// ---- MTCS/Common/Widgets/OperatingButtonWidget.TcPOU
FUNCTION_BLOCK OperatingButtonWidget
VAR_INPUT
END_VAR
VAR_OUTPUT
    text : STRING;
    deactivate : BOOL;
END_VAR
VAR_IN_OUT
    status : OperatingStatus;
	process : ChangeOperatingStateProcess;
END_VAR
VAR
    do_request : BOOL := FALSE;
END_VAR

IF status.auto THEN
    text := 'Manual';
    process.set.state := OperatingStates.MANUAL;
    deactivate := process.statuses.enabledStatus.disabled;
ELSIF status.manual THEN
    text := 'Auto';
    process.set.state := OperatingStates.AUTO;
    deactivate := process.statuses.enabledStatus.disabled;
ELSE
    text := 'Auto';
    process.set.state := OperatingStates.MANUAL;
    deactivate := TRUE;
END_IF


IF do_request THEN
    process.request(state := process.set.state);
    do_request := FALSE;
END_IF

END_FUNCTION_BLOCK

// ---- MTCS/Common/Widgets/LockingButtonWidget.TcPOU
FUNCTION_BLOCK LockingButtonWidget
VAR_INPUT
END_VAR
VAR_OUTPUT
    text : STRING;
    deactivate : BOOL;
END_VAR
VAR_IN_OUT
    status : InitializationStatus;
	lock : Process;
	unlock : Process;
END_VAR
VAR
    do_request : BOOL := FALSE;
END_VAR

IF status.locked THEN
    text := 'Unlock';
    deactivate := unlock.statuses.enabledStatus.disabled;
    
    IF do_request THEN
        unlock.request();
        do_request := FALSE;
    END_IF

ELSIF status.initialized THEN
    text := 'Lock';
    deactivate := lock.statuses.enabledStatus.disabled;
    
    IF do_request THEN
        lock.request();
        do_request := FALSE;
    END_IF
ELSE
    text := 'Unlock';
    deactivate := TRUE;
    do_request := FALSE;
END_IF

END_FUNCTION_BLOCK

// ---- MTCS/Common/HelperCode/SystemToColor.TcPOU
FUNCTION SystemToColor : StatusColor
VAR_IN_OUT
    healthStatus : HealthStatus;
    busyStatus   : BusyStatus;
    initializationStatus : InitializationStatus;
    operatingStatus : OperatingStatus;
END_VAR
VAR_OUTPUT
END_VAR
VAR
END_VAR

IF initializationStatus.shutdown THEN
    SystemToColor.fg := Colors.BLACK;
    SystemToColor.bg := Colors.GRAY;
ELSIF initializationStatus.initializing THEN
    SystemToColor.fg := Colors.WHITE;
    SystemToColor.bg := Colors.BLUE;
ELSE
    IF healthStatus.good THEN
        IF busyStatus.busy THEN
            SystemToColor.fg := Colors.WHITE;
            SystemToColor.bg := Colors.BLUE;
        ELSE
            IF initializationStatus.locked OR operatingStatus.manual THEN
                SystemToColor.fg := Colors.WHITE;
                SystemToColor.bg := Colors.ORANGE;
            ELSE
                SystemToColor.fg := Colors.BLACK;
                SystemToColor.bg := Colors.GREEN;
			END_IF
        END_IF
    ELSIF healthStatus.bad THEN
        SystemToColor.fg := Colors.WHITE;
        SystemToColor.bg := Colors.RED;
    ELSIF healthStatus.warning THEN
        SystemToColor.fg := Colors.WHITE;
        SystemToColor.bg := Colors.ORANGE;
    ELSE
        SystemToColor.fg := Colors.BLACK;
        SystemToColor.bg := Colors.GRAY;
    END_IF
END_IF

END_FUNCTION

// ---- MTCS/Common/HelperCode/BusyToColor.TcPOU
FUNCTION BusyToColor : StatusColor
VAR_IN_OUT
    busyStatus : BusyStatus;
END_VAR
VAR_OUTPUT
END_VAR
VAR
END_VAR

IF busyStatus.idle THEN
    BusyToColor.fg := Colors.BLACK;
    BusyToColor.bg := Colors.GREEN;
ELSIF busyStatus.busy THEN
	BusyToColor.fg := Colors.WHITE;
	BusyToColor.bg := Colors.BLUE;
ELSE
	BusyToColor.fg := Colors.BLACK;
	BusyToColor.bg := Colors.GRAY;
END_IF

END_FUNCTION

// ---- MTCS/Common/HelperCode/DegToRad.TcPOU
FUNCTION DegToRad : LREAL
VAR_INPUT
    degrees : LREAL;
END_VAR
VAR
END_VAR

DegToRad := degrees / 180.0 * PI;

END_FUNCTION

// ---- MTCS/Common/HelperCode/MeasurementToString.TcPOU
FUNCTION_BLOCK MeasurementToString
VAR_INPUT
    value : LREAL;
    format : STRING;
    overrange : BOOL;
    underrange: BOOL;
    error : BOOL;
END_VAR
VAR_OUTPUT
    display : STRING;
    actualStatus : STRING;
END_VAR
VAR_IN_OUT
    alarmStatus : HiHiLoLoAlarmStatus;
    enabledStatus : EnabledStatus;
END_VAR
VAR
    _formatString : FB_FormatString;
END_VAR

// update the display and actualStatus
IF enabledStatus.enabled THEN
    IF overrange THEN
        display := '';
        actualStatus := 'Overrange';
    ELSIF underrange THEN
        display := '';
        actualStatus := 'Underrange';
    ELSIF error THEN
        display := '';
        actualStatus := 'Error';
    ELSE
        // update display:
        _formatString(sFormat := format, 
                      arg1    := F_LREAL(value),
                      sOut    => display);
        // update actualStatus:
        IF alarmStatus.disabled THEN
            actualStatus := 'Valid';
        ELSIF alarmStatus.ok THEN
            actualStatus := 'Valid and within range';
        ELSIF alarmStatus.hi THEN
            actualStatus := 'High!';
        ELSIF alarmStatus.hiHi THEN
            actualStatus := 'Critically high!';
        ELSIF alarmStatus.lo THEN
            actualStatus := 'Low!';
        ELSIF alarmStatus.loLo THEN
            actualStatus := 'Critically low!';
        ELSE
            actualStatus := display;
        END_IF
    END_IF
ELSIF enabledStatus.disabled THEN
    display := '';
    actualStatus := 'Disabled';
ELSE
    display := '';
    actualStatus := 'UNKNOWN';
END_IF

END_FUNCTION_BLOCK

// ---- MTCS/Common/HelperCode/MeasurementToStatus.TcPOU
FUNCTION_BLOCK MeasurementToStatus
VAR_INPUT
    overrange : BOOL;
    underrange: BOOL;
    error : BOOL;
END_VAR
VAR_OUTPUT
    actualStatus : STRING;
END_VAR
VAR_IN_OUT
    alarmStatus : HiHiLoLoAlarmStatus;
    enabledStatus : EnabledStatus;
END_VAR
VAR
END_VAR

// update the display and actualStatus
IF enabledStatus.enabled THEN
    IF overrange THEN
        actualStatus := 'Overrange';
    ELSIF underrange THEN
        actualStatus := 'Underrange';
    ELSIF error THEN
        actualStatus := 'Error';
    ELSE
        // update actualStatus:
        IF alarmStatus.disabled THEN
            actualStatus := 'Valid';
        ELSIF alarmStatus.ok THEN
            actualStatus := 'Valid and within range';
        ELSIF alarmStatus.hi THEN
            actualStatus := 'High!';
        ELSIF alarmStatus.hiHi THEN
            actualStatus := 'Critically high!';
        ELSIF alarmStatus.lo THEN
            actualStatus := 'Low!';
        ELSIF alarmStatus.loLo THEN
            actualStatus := 'Critically low!';
        ELSE
            actualStatus := 'UNKNOWN';
        END_IF
    END_IF
ELSIF enabledStatus.disabled THEN
    actualStatus := 'Disabled';
ELSE
    actualStatus := 'UNKNOWN';
END_IF

END_FUNCTION_BLOCK

// ---- MTCS/Common/HelperCode/RadToDeg.TcPOU
FUNCTION RadToDeg : LREAL
VAR_INPUT
    radians : LREAL;
END_VAR
VAR
END_VAR

RadToDeg := radians / PI * 180.0;

END_FUNCTION

// ---- MTCS/Common/StateMachines/AngularVelocity.TcPOU
FUNCTION_BLOCK AngularVelocity EXTENDS SM_AngularVelocity
VAR_INPUT
END_VAR
VAR_OUTPUT
END_VAR
VAR
    _testVar : INT;
END_VAR

SUPER^();

END_FUNCTION_BLOCK

// ---- MTCS/Common/StateMachines/AngularAcceleration.TcPOU
FUNCTION_BLOCK AngularAcceleration EXTENDS SM_AngularAcceleration
VAR_INPUT
END_VAR
VAR_OUTPUT
END_VAR
VAR
    _testVar : INT;
END_VAR

SUPER^();

END_FUNCTION_BLOCK

// ---- MTCS/Common/StateMachines/AverageCurrent.TcPOU
FUNCTION_BLOCK AverageCurrent EXTENDS SM_AverageCurrent
VAR_INPUT
    noOfSamples : UINT := 100;
    ctrlTimeMultiplier : UINT := 1;
END_VAR
VAR_OUTPUT
END_VAR
VAR
    _ctrl_moving_avg : FB_CTRL_MOVING_AVERAGE;
    _params : ST_CTRL_MOVING_AVERAGE_PARAMS;
    _array : ARRAY [1..100] OF LREAL;
END_VAR

_params.nSamplesToFilter  := noOfSamples;
_params.tCtrlCycleTime    := GLOBAL.config.PLC_CTRL_TIME * ctrlTimeMultiplier;

_ctrl_moving_avg(
    fIn             := SUPER^.newAmpsValue,
    fManSyncValue   := 0.0,
    bSync           := FALSE,
    eMode           := E_CTRL_MODE.eCTRL_MODE_ACTIVE,
    bHold           := FALSE,
    stParams        := _params);

SUPER^(newAmpsValue := _ctrl_moving_avg.fOut);

METHOD FB_init : BOOL
VAR_INPUT
	bInitRetains : BOOL; // if TRUE, the retain variables are initialized (warm start / cold start)
	bInCopyCode : BOOL;  // if TRUE, the instance afterwards gets moved into the copy code (online change)
END_VAR
_params.tTaskCycleTime    := GLOBAL.config.PLC_TASK_TIME;
_params.pWorkArray_ADR    := ADR(_array);
_params.nWorkArray_SIZEOF := SIZEOF(_array);
END_METHOD

END_FUNCTION_BLOCK

// ---- MTCS/Common/StateMachines/AX52XXDrive.TcPOU
FUNCTION_BLOCK AX52XXDrive EXTENDS SM_AX52XXDrive
VAR_INPUT
END_VAR
VAR_OUTPUT
END_VAR
VAR
    _internal : INT; // if no variable is present, the symbols of the superclass are not visible in the OPC UA address space
END_VAR

SUPER^();

END_FUNCTION_BLOCK

// ---- MTCS/Common/StateMachines/BaseProcess.TcPOU
FUNCTION_BLOCK BaseProcess EXTENDS SM_BaseProcess (* default process *)
VAR_INPUT
	_state : INT; // internal state, may or may not be used
END_VAR
VAR_OUTPUT
END_VAR
VAR
END_VAR

// we make it easy for ourselves: every time the process is idle, we reset the startedStatus
IF statuses.busyStatus.idle THEN
	statuses.startedStatus(isStarted := FALSE);
END_IF

_update();

METHOD isIdle : BOOL
VAR_INPUT
END_VAR
isIdle := statuses.busyStatus.idle;
END_METHOD

METHOD _update
VAR_INPUT
END_VAR

IF actualStatus = '' THEN
    IF statuses.enabledStatus.disabled THEN
        actualStatus := '';
    ELSIF statuses.enabledStatus.enabled THEN
        IF statuses.healthStatus.good THEN
            IF statuses.busyStatus.busy THEN
                actualStatus := 'Busy';
            ELSIF statuses.busyStatus.idle THEN
                actualStatus := 'Idle';
            ELSE
                actualStatus := 'Good but UNKNOWN';
            END_IF
        ELSIF statuses.healthStatus.bad THEN
            IF statuses.busyStatus.busy THEN
                actualStatus := 'Error (busy)';
            ELSIF statuses.busyStatus.idle THEN
                actualStatus := 'Error';
            ELSE
                actualStatus := 'Bad but UNKNOWN';
            END_IF
        END_IF
    END_IF
END_IF

SUPER^();
END_METHOD

METHOD setBad
VAR_INPUT
END_VAR
statuses.healthStatus(isGood := FALSE);
END_METHOD

METHOD resetIfIdle
VAR_INPUT
END_VAR
IF statuses.busyStatus.idle  THEN
    
    statuses.healthStatus(isGood := TRUE, hasWarning := FALSE);
    setActualStatus('Idle');
    setFinished();
    
END_IF
END_METHOD

METHOD setBusy
VAR_INPUT
END_VAR
statuses.busyStatus(isBusy := TRUE);
END_METHOD

METHOD setFinished
VAR_INPUT
END_VAR
statuses.busyStatus(isBusy := FALSE);
statuses.startedStatus(isStarted := FALSE);
END_METHOD

METHOD setStarted
VAR_INPUT
END_VAR
statuses.startedStatus(isStarted := TRUE);
END_METHOD

METHOD isBusy : BOOL
VAR_INPUT
END_VAR
isBusy := statuses.busyStatus.busy;
END_METHOD

METHOD setActualStatus
VAR_INPUT
    msg : STRING;
END_VAR
actualStatus := msg;
END_METHOD

METHOD reset
VAR_INPUT
END_VAR
statuses.healthStatus(isGood := TRUE, hasWarning := FALSE);
statuses.busyStatus(isBusy := FALSE);
setActualStatus('Idle');
setFinished();
END_METHOD

METHOD setGood
VAR_INPUT
END_VAR
statuses.healthStatus(isGood := TRUE);
END_METHOD

METHOD isGood : BOOL
VAR_INPUT
END_VAR
isGood := statuses.healthStatus.good;
END_METHOD

METHOD FB_init : BOOL
VAR_INPUT
	bInitRetains : BOOL; // if TRUE, the retain variables are initialized (warm start / cold start)
	bInCopyCode : BOOL;  // if TRUE, the instance afterwards gets moved into the copy code (online change)
END_VAR
statuses.busyStatus(isBusy := FALSE);
statuses.startedStatus(isStarted := FALSE);
statuses.healthStatus(isGood := TRUE);
END_METHOD

METHOD isStarted : BOOL
VAR_INPUT
END_VAR
isStarted := statuses.startedStatus.started;
END_METHOD

END_FUNCTION_BLOCK

// ---- MTCS/Common/StateMachines/BaseXmlDataSrvProcess.TcPOU
FUNCTION_BLOCK BaseXmlDataSrvProcess EXTENDS SM_BaseMcProcess
VAR_INPUT
END_VAR
VAR_OUTPUT
END_VAR
VAR
	testVar3 : BOOL;
END_VAR

SUPER^();

END_FUNCTION_BLOCK

// ---- MTCS/Common/StateMachines/CANopenBus.TcPOU
FUNCTION_BLOCK CANopenBus EXTENDS SM_CANopenBus
VAR_INPUT
END_VAR
VAR_OUTPUT
END_VAR
VAR
    testVar : INT;
END_VAR

//IF GLOBAL.CONFIG.SIMULATION_ACTIVE THEN
//    SUPER^.infoData := 8;
//    SUPER^.wcState := FALSE;
//END_IF

SUPER^();

IF error = 0 THEN
    actualStatus := 'No errors';
ELSE
    actualStatus := CONCAT(USINT_TO_STRING(error), ' boxes have errors');
END_IF

END_FUNCTION_BLOCK

// ---- MTCS/Common/StateMachines/CurrentMeasurement.TcPOU
FUNCTION_BLOCK CurrentMeasurement EXTENDS SM_CurrentMeasurement
VAR_INPUT
END_VAR
VAR_OUTPUT
END_VAR
VAR
    testVar : INT;
END_VAR

SUPER^();

END_FUNCTION_BLOCK

// ---- MTCS/Common/StateMachines/GForce.TcPOU
FUNCTION_BLOCK GForce EXTENDS SM_GForce
VAR_INPUT
END_VAR
VAR_OUTPUT
END_VAR
VAR
    _testVar : INT;
END_VAR

SUPER^();

END_FUNCTION_BLOCK

// ---- MTCS/Common/StateMachines/LinearPositionMeasurement16.TcPOU
FUNCTION_BLOCK LinearPositionMeasurement16 EXTENDS SM_LinearPositionMeasurement16
VAR_INPUT
END_VAR
VAR_OUTPUT
END_VAR
VAR
    noOfSamples : UINT := 100;
    _toStatus : MeasurementToStatus;
	_executeMovingAverage : BOOL;
    _ctrl_moving_avg : FB_CTRL_MOVING_AVERAGE;
    _params : ST_CTRL_MOVING_AVERAGE_PARAMS;
    _array : ARRAY [1..100] OF LREAL;
END_VAR

SUPER^(config := config);

_params.nSamplesToFilter  := noOfSamples;
_params.tCtrlCycleTime    := GLOBAL.config.PLC_CTRL_TIME;

// only call the _ctrl_moving_avg FB once per task cycle (not once every time the xxxMeasurement FB is called)
IF _executeMovingAverage <> GLOBAL.config.PLC_TASK_FLIP THEN
	_executeMovingAverage := GLOBAL.config.PLC_TASK_FLIP;
	_ctrl_moving_avg(
		fIn             := actual.millimeters.value,
		fManSyncValue   := 0.0,
		bSync           := FALSE,
		eMode           := E_CTRL_MODE.eCTRL_MODE_ACTIVE,
		bHold           := FALSE,
		stParams        := _params);
END_IF

// update the average value
average(newMillimetersValue := _ctrl_moving_avg.fOut);
	
_toStatus(
    overrange     := overrange,
    underrange    := underrange,
    error         := error,
    alarmStatus   := statuses.alarmStatus,
    enabledStatus := statuses.enabledStatus,
    actualStatus  => actualStatus);
	
SUPER^(config := config);

METHOD FB_init : BOOL
VAR_INPUT
	bInitRetains : BOOL; // if TRUE, the retain variables are initialized (warm start / cold start)
	bInCopyCode : BOOL;  // if TRUE, the instance afterwards gets moved into the copy code (online change)
END_VAR
_params.tTaskCycleTime    := GLOBAL.config.PLC_TASK_TIME;
_params.pWorkArray_ADR    := ADR(_array);
_params.nWorkArray_SIZEOF := SIZEOF(_array);
END_METHOD

END_FUNCTION_BLOCK

// ---- MTCS/Common/StateMachines/EtherCatDevice.TcPOU
FUNCTION_BLOCK EtherCatDevice EXTENDS SM_EtherCatDevice
VAR_INPUT
END_VAR
VAR_OUTPUT
END_VAR
VAR
    testVar : INT;
END_VAR

IF GLOBAL.CONFIG.SIMULATION_ACTIVE THEN
    SUPER^.infoData := 8;
    SUPER^.wcState := FALSE;
END_IF

SUPER^();

actualStatus := F_ConvStateToString(UINT_TO_WORD(infoData));

END_FUNCTION_BLOCK

// ---- MTCS/Common/StateMachines/FaulhaberDrive.TcPOU
FUNCTION_BLOCK FaulhaberDrive EXTENDS SM_FaulhaberDrive
VAR_INPUT
END_VAR
VAR_OUTPUT
END_VAR
VAR
    _sdoRead : ADSREAD;
    _sdoWrite : ADSWRITE;
    
    noOfWrites : INT := 0;
    
    _currentInitializingState : INT;
END_VAR

SUPER^(config := config);

_initializing();
_sdoReading();
_sdoWriting();

SUPER^(config := config);

METHOD _initializing_write4Bytes
VAR_INPUT
    index : UINT;
    subIndex : USINT;
    value : UDINT;
END_VAR
IF processes.write.isIdle() THEN
    
    processes.write.start(
        index := index, 
        subindex := subIndex, 
        noOfBytes := 4, 
        value1Byte := 0, 
        value2Bytes := 0, 
        value4Bytes := value);
           
    _currentInitializingState := _currentInitializingState + 1;

END_IF
END_METHOD

METHOD _initializing
VAR_INPUT    

END_VAR
VAR
END_VAR
IF processes.initialize.statuses.busyStatus.busy THEN
    
    IF processes.initialize.statuses.startedStatus.notStarted THEN
        IF config.sendAtInitialization THEN
            _currentInitializingState := 0;
        ELSE
            _currentInitializingState := 1000;
		END_IF
        processes.initialize.setStarted();
	END_IF

    CASE _currentInitializingState OF
        
        0:
            _initializing_write1Byte(index := 16#6060, subindex := 0, value := config.modesOfOperation);
        1:
            _initializing_waitForWrite();
        2:
            _initializing_write1Byte(index := 16#607E, subindex := 0, value := config.polarity);
        3:
            _initializing_waitForWrite();
        4:
            _initializing_write4Bytes(index := 16#607F, subindex := 0, value := config.maxProfileVelocity);
        5:
            _initializing_waitForWrite();
        6:
            _initializing_write1Byte(index := 16#2310, subindex := 1, value := config.negativeLimitSwitch);
        7:
            _initializing_waitForWrite();
        8:
            _initializing_write1Byte(index := 16#2310, subindex := 2, value := config.positiveLimitSwitch);
        9:
            _initializing_waitForWrite();
        10:
            _initializing_write1Byte(index := 16#2310, subindex := 3, value := config.homingSwitch);
        11:
            _initializing_waitForWrite();
        12:
            _initializing_write1Byte(index := 16#2310, subindex := 5, value := config.limitSwitchPolarity);
        13:
            _initializing_waitForWrite();
        14:
            _initializing_write2Bytes(index := 16#2333, subindex := 1, value := config.continuousCurrentLimit);
        15:
            _initializing_waitForWrite();
        16:
            _initializing_write2Bytes(index := 16#2333, subindex := 2, value := config.peakCurrentLimit);
        17:
            _initializing_waitForWrite();
        18:
            _initializing_write2Bytes(index := 16#2331, subindex := 1, value := config.velocityControlProportionalTerm);
        19:
            _initializing_waitForWrite();
        20:
            _initializing_write2Bytes(index := 16#2331, subindex := 2, value := config.velocityControlIntegralTerm);
        21:
            _initializing_waitForWrite();
        22:
            // just finish!
            _currentInitializingState := 1000;
        999:
            // error!
            processes.initialize.setBad();
            processes.initialize.setFinished();
        1000:
            // all done!
            processes.initialize.setGood();
            processes.initialize.setFinished();
	END_CASE

END_IF
END_METHOD

METHOD configure
VAR_INPUT
    noOfCurrentSamples : UINT;
    ctrlTimeMultiplier : UINT;
END_VAR
averageCurrent.ctrlTimeMultiplier := ctrlTimeMultiplier;
averageCurrent.noOfSamples := noOfCurrentSamples;
END_METHOD

METHOD _initializing_write1Byte
VAR_INPUT
    index : UINT;
    subIndex : USINT;
    value : USINT;
END_VAR
IF processes.write.isIdle() THEN
    
    processes.write.start(
        index := index, 
        subindex := subIndex, 
        noOfBytes := 1, 
        value1Byte := value, 
        value2Bytes := 0, 
        value4Bytes := 0);

    _currentInitializingState := _currentInitializingState + 1;
        
END_IF
END_METHOD

METHOD _initializing_write2Bytes
VAR_INPUT
    index : UINT;
    subIndex : USINT;
    value : UINT;
END_VAR
IF processes.write.isIdle() THEN
    
    processes.write.start(
        index := index, 
        subindex := subIndex, 
        noOfBytes := 2, 
        value1Byte := 0, 
        value2Bytes := value, 
        value4Bytes := 0);

    _currentInitializingState := _currentInitializingState + 1;
            
END_IF
END_METHOD

METHOD _initializing_waitForWrite
VAR_INPUT
END_VAR
IF processes.write.isIdle() THEN
    IF processes.write.isGood() THEN
        _currentInitializingState := _currentInitializingState + 1;
    ELSE
        _currentInitializingState := 999;
    END_IF
END_IF
END_METHOD

METHOD _sdoWriting
VAR_INPUT
END_VAR
VAR
    srcAddress : PVOID;
END_VAR
IF processes.write.statuses.busyStatus.busy THEN
    
    IF processes.write.get.noOfBytes = 1 THEN
        srcAddress := ADR(processes.write.get.value1Byte);
        processes.write.setGood();
    ELSIF processes.write.get.noOfBytes = 2 THEN
        srcAddress := ADR(processes.write.get.value2Bytes);
        processes.write.setGood();
    ELSIF processes.write.get.noOfBytes = 4 THEN
        srcAddress := ADR(processes.write.get.value4Bytes);
        processes.write.setGood();
    ELSE
        processes.write.setBad();
        processes.write.setFinished();
	END_IF
     
    
    IF processes.write.statuses.healthStatus.good THEN
         
        IF NOT processes.write.statuses.startedStatus.started THEN
        
            noOfWrites := noOfWrites + 1;
            
            (* Make sure the Execute input is reset *)
            _sdoWrite(WRITE := FALSE);
        
            (* execute the SDO read command *)
            _sdoWrite(
                 NETID      := config.CANopenBusNetId,
                 PORT       := config.CANopenNodePort,
                 IDXGRP     := processes.write.get.index,
                 IDXOFFS    := processes.write.get.subindex,
                 SRCADDR    := srcAddress,
                 LEN        := processes.write.get.noOfBytes,
                 WRITE      := TRUE);
            
             processes.write.setStarted();
        ELSE
            (* Make sure the Execute input is reset *)
            _sdoWrite(WRITE := FALSE);
            
            (* update the health status *)
            SUPER^.processes.write.statuses.healthStatus(isGood := NOT _sdoWrite.ERR);
            
            (* update the busy status *)
            SUPER^.processes.write.statuses.busyStatus(isBusy := _sdoWrite.BUSY);
            
            (* update the error ID *)
            SUPER^.processes.write.errorId := _sdoWrite.ERRID;
		END_IF
        
             
	END_IF
    

 
END_IF
END_METHOD

METHOD _sdoReading
VAR_INPUT
END_VAR
VAR
    valueAddress : PVOID;
END_VAR
IF processes.read.statuses.busyStatus.busy THEN
    
    IF processes.read.get.noOfBytes = 1 THEN
        valueAddress := ADR(processes.read.value1Byte);
        processes.read.setGood();
    ELSIF processes.read.get.noOfBytes = 2 THEN
        valueAddress := ADR(processes.read.value2Bytes);
        processes.read.setGood();
    ELSIF processes.read.get.noOfBytes = 4 THEN
        valueAddress := ADR(processes.read.value4Bytes);
        processes.read.setGood();
    ELSE
        processes.read.setBad();
        processes.read.setFinished();
	END_IF
     
    
    IF processes.read.statuses.healthStatus.good THEN
         
        IF NOT processes.read.statuses.startedStatus.started THEN
            _sdoRead(READ   := FALSE);
            
            (* execute the SDO read command *)
            _sdoRead(
                 NETID      := config.CANopenBusNetId,
                 PORT       := config.CANopenNodePort,
                 IDXGRP     := processes.read.get.index,
                 IDXOFFS    := processes.read.get.subindex,
                 DESTADDR   := valueAddress,
                 LEN        := processes.read.get.noOfBytes,
                 READ       := TRUE);
            
             processes.read.setStarted();
             
		END_IF
        
       (* Make sure the Execute input is reset *)
       //_sdoRead(bExecute   := FALSE);
        _sdoRead(READ   := FALSE);
        
        (* update the health status *)
        SUPER^.processes.read.statuses.healthStatus(isGood := NOT _sdoRead.ERR);
        
        (* update the busy status *)
        SUPER^.processes.read.statuses.busyStatus(isBusy := _sdoRead.BUSY);
        
        (* update the error ID *)
        SUPER^.processes.read.errorId := _sdoRead.ERRID;
             
	END_IF
    

 
END_IF
END_METHOD

END_FUNCTION_BLOCK

// ---- MTCS/Common/StateMachines/ForceMeasurement.TcPOU
FUNCTION_BLOCK ForceMeasurement EXTENDS SM_ForceMeasurement
VAR_INPUT
END_VAR
VAR_OUTPUT
END_VAR
VAR
    noOfSamples : UINT := 100;
    _toStatus : MeasurementToStatus;
	_executeMovingAverage : BOOL;
    _ctrl_moving_avg : FB_CTRL_MOVING_AVERAGE;
    _params : ST_CTRL_MOVING_AVERAGE_PARAMS;
    _array : ARRAY [1..100] OF LREAL;
END_VAR

SUPER^(config := config);

_params.nSamplesToFilter  := noOfSamples;
_params.tCtrlCycleTime    := GLOBAL.config.PLC_CTRL_TIME;

// only call the _ctrl_moving_avg FB once per task cycle (not once every time the xxxMeasurement FB is called)
IF _executeMovingAverage <> GLOBAL.config.PLC_TASK_FLIP THEN
	_executeMovingAverage := GLOBAL.config.PLC_TASK_FLIP;
	_ctrl_moving_avg(
		fIn             := actual.newton.value,
		fManSyncValue   := 0.0,
		bSync           := FALSE,
		eMode           := E_CTRL_MODE.eCTRL_MODE_ACTIVE,
		bHold           := FALSE,
		stParams        := _params);
END_IF

// update the average value
average(newNewtonValue := _ctrl_moving_avg.fOut);
	
_toStatus(
    overrange     := overrange,
    underrange    := underrange,
    error         := error,
    alarmStatus   := statuses.alarmStatus,
    enabledStatus := statuses.enabledStatus,
    actualStatus  => actualStatus);
	
SUPER^(config := config);

METHOD FB_init : BOOL
VAR_INPUT
	bInitRetains : BOOL; // if TRUE, the retain variables are initialized (warm start / cold start)
	bInCopyCode : BOOL;  // if TRUE, the instance afterwards gets moved into the copy code (online change)
END_VAR
_params.tTaskCycleTime    := GLOBAL.config.PLC_TASK_TIME;
_params.pWorkArray_ADR    := ADR(_array);
_params.nWorkArray_SIZEOF := SIZEOF(_array);
END_METHOD

END_FUNCTION_BLOCK

// ---- MTCS/Common/StateMachines/Frequency.TcPOU
FUNCTION_BLOCK Frequency EXTENDS SM_Frequency
VAR_INPUT
END_VAR
VAR_OUTPUT
END_VAR
VAR
    _testVar : INT;
END_VAR

SUPER^();

END_FUNCTION_BLOCK

// ---- MTCS/Common/StateMachines/FrequencyMeasurement.TcPOU
FUNCTION_BLOCK FrequencyMeasurement EXTENDS SM_FrequencyMeasurement
VAR_INPUT
END_VAR
VAR_OUTPUT
END_VAR
VAR
    noOfSamples : UINT := 100;
    _toStatus : MeasurementToStatus;
	_executeMovingAverage : BOOL;
    _ctrl_moving_avg : FB_CTRL_MOVING_AVERAGE;
    _params : ST_CTRL_MOVING_AVERAGE_PARAMS;
    _array : ARRAY [1..100] OF LREAL;
END_VAR

SUPER^(config := config);

_params.nSamplesToFilter  := noOfSamples;
_params.tCtrlCycleTime    := GLOBAL.config.PLC_CTRL_TIME;

// only call the _ctrl_moving_avg FB once per task cycle (not once every time the xxxMeasurement FB is called)
IF _executeMovingAverage <> GLOBAL.config.PLC_TASK_FLIP THEN
	_executeMovingAverage := GLOBAL.config.PLC_TASK_FLIP;
	_ctrl_moving_avg(
		fIn             := actual.hertz.value,
		fManSyncValue   := 0.0,
		bSync           := FALSE,
		eMode           := E_CTRL_MODE.eCTRL_MODE_ACTIVE,
		bHold           := FALSE,
		stParams        := _params);
END_IF

// update the average value
average(newHertzValue := _ctrl_moving_avg.fOut);
	
_toStatus(
    overrange     := overrange,
    underrange    := underrange,
    error         := error,
    alarmStatus   := statuses.alarmStatus,
    enabledStatus := statuses.enabledStatus,
    actualStatus  => actualStatus);
	
SUPER^(config := config);

METHOD FB_init : BOOL
VAR_INPUT
	bInitRetains : BOOL; // if TRUE, the retain variables are initialized (warm start / cold start)
	bInCopyCode : BOOL;  // if TRUE, the instance afterwards gets moved into the copy code (online change)
END_VAR
_params.tTaskCycleTime    := GLOBAL.config.PLC_TASK_TIME;
_params.pWorkArray_ADR    := ADR(_array);
_params.nWorkArray_SIZEOF := SIZEOF(_array);
END_METHOD

END_FUNCTION_BLOCK

// ---- MTCS/Common/StateMachines/Fraction.TcPOU
FUNCTION_BLOCK Fraction EXTENDS SM_Fraction
VAR_INPUT
END_VAR
VAR_OUTPUT
END_VAR
VAR
    _testVar_Fraction : BOOL;
END_VAR

SUPER^();

END_FUNCTION_BLOCK

// ---- MTCS/Common/StateMachines/LinearAxis.TcPOU
FUNCTION_BLOCK LinearAxis EXTENDS SM_LinearAxis;
VAR_INPUT
END_VAR
VAR_OUTPUT
END_VAR
VAR
    _testVar_LinearAxis : BOOL;
END_VAR

SUPER^();

END_FUNCTION_BLOCK

// ---- MTCS/Common/StateMachines/LinearPosition.TcPOU
FUNCTION_BLOCK LinearPosition EXTENDS SM_LinearPosition
VAR_INPUT
END_VAR
VAR_OUTPUT
END_VAR
VAR
    _testVar_LinearPosition : INT;
END_VAR

SUPER^();

// do stuff

//SUPER^();

END_FUNCTION_BLOCK

// ---- MTCS/Common/StateMachines/LinearPositionMeasurementU32.TcPOU
FUNCTION_BLOCK LinearPositionMeasurementU32 EXTENDS SM_LinearPositionMeasurementU32
VAR_INPUT
    noOfSamples : UINT := 100;
END_VAR
VAR_OUTPUT
END_VAR
VAR
    _toStatus : MeasurementToStatus;
	_executeMovingAverage : BOOL;
    _ctrl_moving_avg : FB_CTRL_MOVING_AVERAGE;
    _params : ST_CTRL_MOVING_AVERAGE_PARAMS;
    _array : ARRAY [1..100] OF LREAL;
END_VAR

SUPER^(config := config);

_params.nSamplesToFilter  := noOfSamples;
_params.tCtrlCycleTime    := GLOBAL.config.PLC_CTRL_TIME;

// only call the _ctrl_moving_avg FB once per task cycle (not once every time the xxxMeasurement FB is called)
IF _executeMovingAverage <> GLOBAL.config.PLC_TASK_FLIP THEN
	_executeMovingAverage := GLOBAL.config.PLC_TASK_FLIP;
	_ctrl_moving_avg(
		fIn             := actual.millimeters.value,
		fManSyncValue   := 0.0,
		bSync           := FALSE,
		eMode           := E_CTRL_MODE.eCTRL_MODE_ACTIVE,
		bHold           := FALSE,
		stParams        := _params);
END_IF

// update the average value
average(newMillimetersValue := _ctrl_moving_avg.fOut);
	
_toStatus(
    overrange     := overrange,
    underrange    := underrange,
    error         := error,
    alarmStatus   := statuses.alarmStatus,
    enabledStatus := statuses.enabledStatus,
    actualStatus  => actualStatus);
	
SUPER^(config := config);

METHOD FB_init : BOOL
VAR_INPUT
	bInitRetains : BOOL; // if TRUE, the retain variables are initialized (warm start / cold start)
	bInCopyCode : BOOL;  // if TRUE, the instance afterwards gets moved into the copy code (online change)
END_VAR
_params.tTaskCycleTime    := GLOBAL.config.PLC_TASK_TIME;
_params.pWorkArray_ADR    := ADR(_array);
_params.nWorkArray_SIZEOF := SIZEOF(_array);
END_METHOD

END_FUNCTION_BLOCK

// ---- MTCS/Common/StateMachines/LinearVelocity.TcPOU
FUNCTION_BLOCK LinearVelocity EXTENDS SM_LinearVelocity
VAR_INPUT
END_VAR
VAR_OUTPUT
END_VAR
VAR
    testVar : INT;
END_VAR

SUPER^();

END_FUNCTION_BLOCK

// ---- MTCS/Common/StateMachines/PressureMeasurement.TcPOU
FUNCTION_BLOCK PressureMeasurement EXTENDS SM_PressureMeasurement
VAR_INPUT
END_VAR
VAR_OUTPUT
END_VAR
VAR
    noOfSamples : UINT := 100;
    _toStatus : MeasurementToStatus;
	_executeMovingAverage : BOOL;
    _ctrl_moving_avg : FB_CTRL_MOVING_AVERAGE;
    _params : ST_CTRL_MOVING_AVERAGE_PARAMS;
    _array : ARRAY [1..100] OF LREAL;
END_VAR

SUPER^(config := config);

_params.nSamplesToFilter  := noOfSamples;
_params.tCtrlCycleTime    := GLOBAL.config.PLC_CTRL_TIME;

// only call the _ctrl_moving_avg FB once per task cycle (not once every time the xxxMeasurement FB is called)
IF _executeMovingAverage <> GLOBAL.config.PLC_TASK_FLIP THEN
	_executeMovingAverage := GLOBAL.config.PLC_TASK_FLIP;
	_ctrl_moving_avg(
		fIn             := actual.bar.value,
		fManSyncValue   := 0.0,
		bSync           := FALSE,
		eMode           := E_CTRL_MODE.eCTRL_MODE_ACTIVE,
		bHold           := FALSE,
		stParams        := _params);
END_IF

// update the average value
average(newBarValue := _ctrl_moving_avg.fOut);
	
_toStatus(
    overrange     := overrange,
    underrange    := underrange,
    error         := error,
    alarmStatus   := statuses.alarmStatus,
    enabledStatus := statuses.enabledStatus,
    actualStatus  => actualStatus);
    
SUPER^(config := config);

METHOD FB_init : BOOL
VAR_INPUT
	bInitRetains : BOOL; // if TRUE, the retain variables are initialized (warm start / cold start)
	bInCopyCode : BOOL;  // if TRUE, the instance afterwards gets moved into the copy code (online change)
END_VAR
_params.tTaskCycleTime    := GLOBAL.config.PLC_TASK_TIME;
_params.pWorkArray_ADR    := ADR(_array);
_params.nWorkArray_SIZEOF := SIZEOF(_array);
END_METHOD

END_FUNCTION_BLOCK

// ---- MTCS/Common/StateMachines/ProcessStep.TcPOU
FUNCTION_BLOCK ProcessStep EXTENDS SM_ProcessStep
VAR_INPUT
    description : STRING;
END_VAR
VAR_OUTPUT
END_VAR
VAR
END_VAR

SUPER^(process := process);

METHOD isGood : BOOL
VAR_INPUT
END_VAR
isGood := process.isGood();
END_METHOD

METHOD isWarning : BOOL
VAR_INPUT
END_VAR
isWarning := process.statuses.healthStatus.warning;
END_METHOD

METHOD isBusy : BOOL
VAR_INPUT
END_VAR
isBusy := process.isBusy();
END_METHOD

METHOD PUBLIC isBad : BOOL
VAR_INPUT
END_VAR
isBad := process.statuses.healthStatus.bad;
END_METHOD

END_FUNCTION_BLOCK

// ---- MTCS/Common/StateMachines/QuantityValue.TcPOU
FUNCTION_BLOCK QuantityValue EXTENDS SM_QuantityValue
VAR_INPUT
END_VAR
VAR_OUTPUT
END_VAR
VAR
    testVar : INT;
END_VAR

SUPER^();

// do stuff

SUPER^();

END_FUNCTION_BLOCK

// ---- MTCS/Common/StateMachines/RelativeHumidityMeasurement.TcPOU
FUNCTION_BLOCK RelativeHumidityMeasurement EXTENDS SM_RelativeHumidityMeasurement
VAR_INPUT
END_VAR
VAR_OUTPUT
END_VAR
VAR
    _toStatus : MeasurementToStatus;
    noOfSamples : UINT := 100;
	_executeMovingAverage : BOOL;
    _ctrl_moving_avg : FB_CTRL_MOVING_AVERAGE;
    _params : ST_CTRL_MOVING_AVERAGE_PARAMS;
    _array : ARRAY [1..100] OF LREAL;
END_VAR

SUPER^(config := config);

_params.nSamplesToFilter  := noOfSamples;
_params.tCtrlCycleTime    := GLOBAL.config.PLC_CTRL_TIME;

// only call the _ctrl_moving_avg FB once per task cycle (not once every time the xxxMeasurement FB is called)
IF _executeMovingAverage <> GLOBAL.config.PLC_TASK_FLIP THEN
	_executeMovingAverage := GLOBAL.config.PLC_TASK_FLIP;
	_ctrl_moving_avg(
		fIn             := actual.unitless.value,
		fManSyncValue   := 0.0,
		bSync           := FALSE,
		eMode           := E_CTRL_MODE.eCTRL_MODE_ACTIVE,
		bHold           := FALSE,
		stParams        := _params);
END_IF

average(newFractionValue := _ctrl_moving_avg.fOut);

_toStatus(
    overrange     := overrange,
    underrange    := underrange,
    error         := error,
    alarmStatus   := statuses.alarmStatus,
    enabledStatus := statuses.enabledStatus,
    actualStatus  => actualStatus);
    
SUPER^(config := config);

METHOD FB_init : BOOL
VAR_INPUT
	bInitRetains : BOOL; // if TRUE, the retain variables are initialized (warm start / cold start)
	bInCopyCode : BOOL;  // if TRUE, the instance afterwards gets moved into the copy code (online change)
END_VAR
_params.tTaskCycleTime    := GLOBAL.config.PLC_TASK_TIME;
_params.pWorkArray_ADR    := ADR(_array);
_params.nWorkArray_SIZEOF := SIZEOF(_array);
END_METHOD

END_FUNCTION_BLOCK

// ---- MTCS/Common/StateMachines/SimpleRelay.TcPOU
FUNCTION_BLOCK SimpleRelay EXTENDS SM_SimpleRelay
VAR_INPUT
END_VAR
VAR_OUTPUT
END_VAR
VAR
    testVar : INT;
END_VAR

_update();
_switching();
_update();

METHOD _update
VAR_INPUT
END_VAR
SUPER^();

IF digitalOutput THEN
    actualStatus := 'Enabled';
ELSE
    actualStatus := 'Disabled';
END_IF
END_METHOD

METHOD _switching
VAR_INPUT
END_VAR
IF processes.setEnabled.isBusy() THEN
    
    digitalOutput := processes.setEnabled.get.enabled;

    processes.setEnabled.setGood();
    processes.setEnabled.setFinished();
    
END_IF
END_METHOD

END_FUNCTION_BLOCK

// ---- MTCS/Common/StateMachines/SSIEncoder.TcPOU
FUNCTION_BLOCK SSIEncoder EXTENDS SM_SSIEncoder
VAR_INPUT
END_VAR
VAR_OUTPUT
END_VAR
VAR
    _testVar_SSIEncoder : BOOL; // at least one variable is needed to expose this FB via OPC UA
END_VAR

SUPER^();

END_FUNCTION_BLOCK

// ---- MTCS/Common/StateMachines/TemperatureMeasurement.TcPOU
FUNCTION_BLOCK TemperatureMeasurement EXTENDS SM_TemperatureMeasurement
VAR_INPUT
END_VAR
VAR_OUTPUT
END_VAR
VAR
    noOfSamples : UINT := 100;
    _toStatus : MeasurementToStatus;
	_executeMovingAverage : BOOL;
    _ctrl_moving_avg : FB_CTRL_MOVING_AVERAGE;
    _params : ST_CTRL_MOVING_AVERAGE_PARAMS;
    _array : ARRAY [1..100] OF LREAL;
END_VAR

SUPER^(config := config);

_params.nSamplesToFilter  := noOfSamples;
_params.tCtrlCycleTime    := GLOBAL.config.PLC_CTRL_TIME;

// only call the _ctrl_moving_avg FB once per task cycle (not once every time the xxxMeasurement FB is called)
IF _executeMovingAverage <> GLOBAL.config.PLC_TASK_FLIP THEN
	_executeMovingAverage := GLOBAL.config.PLC_TASK_FLIP;
	_ctrl_moving_avg(
		fIn             := actual.celsius.value,
		fManSyncValue   := 0.0,
		bSync           := FALSE,
		eMode           := E_CTRL_MODE.eCTRL_MODE_ACTIVE,
		bHold           := FALSE,
		stParams        := _params);
END_IF

average(newCelsiusValue := _ctrl_moving_avg.fOut);
	
_toStatus(
    overrange     := overrange,
    underrange    := underrange,
    error         := error,
    alarmStatus   := statuses.alarmStatus,
    enabledStatus := statuses.enabledStatus,
    actualStatus  => actualStatus);
	
SUPER^(config := config);

METHOD FB_init : BOOL
VAR_INPUT
	bInitRetains : BOOL; // if TRUE, the retain variables are initialized (warm start / cold start)
	bInCopyCode : BOOL;  // if TRUE, the instance afterwards gets moved into the copy code (online change)
END_VAR
_params.tTaskCycleTime    := GLOBAL.config.PLC_TASK_TIME;
_params.pWorkArray_ADR    := ADR(_array);
_params.nWorkArray_SIZEOF := SIZEOF(_array);
END_METHOD

END_FUNCTION_BLOCK

// ---- MTCS/Common/StateMachines/TorqueLimit.TcPOU
FUNCTION_BLOCK TorqueLimit EXTENDS SM_TorqueLimit
VAR_INPUT
END_VAR
VAR_OUTPUT
END_VAR
VAR
    _testVar : INT;
END_VAR

SUPER^();

END_FUNCTION_BLOCK

// ---- MTCS/Common/StateMachines/Voltage.TcPOU
FUNCTION_BLOCK Voltage EXTENDS SM_Voltage
VAR_INPUT
END_VAR
VAR_OUTPUT
END_VAR
VAR
    _testVar : INT;
END_VAR

SUPER^();

END_FUNCTION_BLOCK

// ---- MTCS/Common/StateMachines/VoltageMeasurement.TcPOU
FUNCTION_BLOCK VoltageMeasurement EXTENDS SM_VoltageMeasurement
VAR_INPUT
END_VAR
VAR_OUTPUT
END_VAR
VAR
    noOfSamples : UINT := 100;
    _toStatus : MeasurementToStatus;
	_executeMovingAverage : BOOL;
    _ctrl_moving_avg : FB_CTRL_MOVING_AVERAGE;
    _params : ST_CTRL_MOVING_AVERAGE_PARAMS;
    _array : ARRAY [1..100] OF LREAL;
END_VAR

SUPER^(config := config);

_params.nSamplesToFilter  := noOfSamples;
_params.tCtrlCycleTime    := GLOBAL.config.PLC_CTRL_TIME;

// only call the _ctrl_moving_avg FB once per task cycle (not once every time the xxxMeasurement FB is called)
IF _executeMovingAverage <> GLOBAL.config.PLC_TASK_FLIP THEN
	_executeMovingAverage := GLOBAL.config.PLC_TASK_FLIP;
	_ctrl_moving_avg(
		fIn             := actual.volt.value,
		fManSyncValue   := 0.0,
		bSync           := FALSE,
		eMode           := E_CTRL_MODE.eCTRL_MODE_ACTIVE,
		bHold           := FALSE,
		stParams        := _params);
END_IF

average(newVoltValue := _ctrl_moving_avg.fOut);

_toStatus(
    overrange     := overrange,
    underrange    := underrange,
    error         := error,
    alarmStatus   := statuses.alarmStatus,
    enabledStatus := statuses.enabledStatus,
    actualStatus  => actualStatus);
    
SUPER^(config := config);

METHOD FB_init : BOOL
VAR_INPUT
	bInitRetains : BOOL; // if TRUE, the retain variables are initialized (warm start / cold start)
	bInCopyCode : BOOL;  // if TRUE, the instance afterwards gets moved into the copy code (online change)
END_VAR
_params.tTaskCycleTime    := GLOBAL.config.PLC_TASK_TIME;
_params.pWorkArray_ADR    := ADR(_array);
_params.nWorkArray_SIZEOF := SIZEOF(_array);
END_METHOD

END_FUNCTION_BLOCK

// ---- MTCS/Common/StateMachines/GForceMeasurement.TcPOU
FUNCTION_BLOCK GForceMeasurement EXTENDS SM_GForceMeasurement
VAR_INPUT
END_VAR
VAR_OUTPUT
END_VAR
VAR
    noOfSamples : UINT := 100;
	_executeMovingAverage : BOOL;
    _ctrl_moving_avg : FB_CTRL_MOVING_AVERAGE;
    _params : ST_CTRL_MOVING_AVERAGE_PARAMS;
    _array : ARRAY [1..100] OF LREAL;
END_VAR

SUPER^();

_params.nSamplesToFilter  := noOfSamples;
_params.tCtrlCycleTime    := GLOBAL.config.PLC_CTRL_TIME;

// only call the _ctrl_moving_avg FB once per task cycle (not once every time the xxxMeasurement FB is called)
IF _executeMovingAverage <> GLOBAL.config.PLC_TASK_FLIP THEN
	_executeMovingAverage := GLOBAL.config.PLC_TASK_FLIP;
	_ctrl_moving_avg(
		fIn             := actual.milliG.value,
		fManSyncValue   := 0.0,
		bSync           := FALSE,
		eMode           := E_CTRL_MODE.eCTRL_MODE_ACTIVE,
		bHold           := FALSE,
		stParams        := _params);
END_IF

average(newMilliGValue := _ctrl_moving_avg.fOut);

IF error THEN
    actualStatus := 'Sensors error'; 
ELSE
    actualStatus := 'Sensors OK';
END_IF
    
SUPER^();

METHOD FB_init : BOOL
VAR_INPUT
	bInitRetains : BOOL; // if TRUE, the retain variables are initialized (warm start / cold start)
	bInCopyCode : BOOL;  // if TRUE, the instance afterwards gets moved into the copy code (online change)
END_VAR
_params.tTaskCycleTime    := GLOBAL.config.PLC_TASK_TIME;
_params.pWorkArray_ADR    := ADR(_array);
_params.nWorkArray_SIZEOF := SIZEOF(_array);
END_METHOD

END_FUNCTION_BLOCK

// ---- MTCS/Common/Widgets/AX52XXDriveWidget.TcPOU
FUNCTION_BLOCK AX52XXDriveWidget
VAR_INPUT
END_VAR
VAR_OUTPUT
END_VAR
VAR_IN_OUT
	ref : AX52XXDrive;
END_VAR
VAR
	actualStatus : StatusWidget;
    channelA : AX52XXDriveChannelWidget;
    channelB : AX52XXDriveChannelWidget;
END_VAR


actualStatus(text  := ref.actualStatus,
             color := HealthBusyToColor(healthStatus := ref.statuses.healthStatus, 
                                        busyStatus   := ref.statuses.busyStatus));
                                        
channelA(ref := ref.parts.channelA, name := 'Channel A');    
channelB(ref := ref.parts.channelB, name := 'Channel B');

END_FUNCTION_BLOCK

// ---- MTCS/Common/Widgets/CANopenBusWidget.TcPOU
FUNCTION_BLOCK CANopenBusWidget
VAR_INPUT
END_VAR
VAR_OUTPUT
END_VAR
VAR
	actualStatus : StatusWidget;
END_VAR
VAR_IN_OUT
	ref : CANopenBus;
END_VAR

actualStatus(text := ref.actualStatus, color := HealthToColor(ref.statuses.healthStatus));

END_FUNCTION_BLOCK

// ---- MTCS/Common/Widgets/EtherCatDeviceWidget.TcPOU
FUNCTION_BLOCK EtherCatDeviceWidget
VAR_INPUT
END_VAR
VAR_OUTPUT
END_VAR
VAR
	actualStatus : StatusWidget;
END_VAR
VAR_IN_OUT
	device : EtherCatDevice;
END_VAR

actualStatus(text  := device.actualStatus, 
             color := HealthToColor(device.statuses.healthStatus));

END_FUNCTION_BLOCK

// ---- MTCS/Common/Widgets/FaulhaberDriveWidget.TcPOU
FUNCTION_BLOCK FaulhaberDriveWidget
VAR_INPUT
    readNoOfBytesRadioButtonItem : INT := 0;
    readNoOfBytes : UDINT;
    writeNoOfBytesRadioButtonItem : INT := 0;
    writeNoOfBytes : UDINT;
END_VAR
VAR_OUTPUT
    readResultValue : UDINT;
END_VAR
VAR_IN_OUT
    ref : FaulhaberDrive;
END_VAR
VAR
	actualStatus : StatusWidget;
	sdoReadStatus : StatusWidget;
	sdoWriteStatus : StatusWidget;
END_VAR

actualStatus(text := ref.actualStatus, 
             color := HealthBusyToColor(healthStatus := ref.statuses.healthStatus, 
                                        busyStatus := ref.statuses.busyStatus));
                                        
sdoReadStatus(text := ref.processes.read.actualStatus,
              color := HealthBusyToColor(healthStatus := ref.processes.read.statuses.healthStatus, 
                                         busyStatus := ref.processes.read.statuses.busyStatus));
sdoWriteStatus(text := ref.processes.write.actualStatus,
               color := HealthBusyToColor(healthStatus := ref.processes.write.statuses.healthStatus, 
                                         busyStatus := ref.processes.write.statuses.busyStatus));

IF readNoOfBytesRadioButtonItem = 0 THEN // first item of the radiobutton is selected
    readNoOfBytes := 1;
    readResultValue := ref.processes.read.value1Byte;
ELSIF readNoOfBytesRadioButtonItem = 1 THEN // second item of the radiobutton is selected
    readNoOfBytes := 2;
    readResultValue := ref.processes.read.value2Bytes;
ELSIF readNoOfBytesRadioButtonItem = 2 THEN // third item of the radiobutton is selected
    readNoOfBytes := 4;
    readResultValue := ref.processes.read.value4Bytes;
END_IF

IF writeNoOfBytesRadioButtonItem = 0 THEN // first item of the radiobutton is selected
    writeNoOfBytes := 1;
ELSIF writeNoOfBytesRadioButtonItem = 1 THEN // second item of the radiobutton is selected
    writeNoOfBytes := 2;
ELSIF writeNoOfBytesRadioButtonItem = 2 THEN // third item of the radiobutton is selected
    writeNoOfBytes := 4;
END_IF

END_FUNCTION_BLOCK

// ---- MTCS/Common/Widgets/ActivityStatusWidget.TcPOU
FUNCTION_BLOCK ActivityStatusWidget
VAR_INPUT
END_VAR
VAR_OUTPUT
	fgColor : DWORD;
	bgColor : DWORD;
	description : STRING;
END_VAR
VAR_IN_OUT
	status : ActivityStatus;
END_VAR
VAR
END_VAR

IF status.sleeping THEN
	fgColor := Colors.BLACK;
	bgColor := Colors.GRAY;
	description := 'Sleeping';
ELSIF status.awake THEN
	fgColor := Colors.BLACK;
	bgColor := Colors.GREEN;
	description := 'Awake';
ELSIF status.moving THEN
	fgColor := Colors.BLACK;
	bgColor := Colors.GREEN;
	description := 'Moving';
ELSE
	fgColor := Colors.BLACK;
	bgColor := Colors.GRAY;
	description := 'Initialize!';
END_IF

END_FUNCTION_BLOCK

// ---- MTCS/Common/Widgets/LinearAxisWidget.TcPOU
FUNCTION_BLOCK LinearAxisWidget
VAR_INPUT
END_VAR
VAR_OUTPUT
    positionSymbol : STRING := 'mm';
    velocitySymbol : STRING := 'mm/s';
END_VAR
VAR_IN_OUT
    baseRef : LinearAxis;
    ref : LinearAxis;
END_VAR
VAR
    base : BaseAxisWidget;
END_VAR

base(ref := baseRef);

END_FUNCTION_BLOCK

// ---- MTCS/Common/Widgets/ActivityButtonWidget.TcPOU
FUNCTION_BLOCK ActivityButtonWidget
VAR_INPUT
END_VAR
VAR_OUTPUT
    text : STRING;
    deactivate : BOOL;
END_VAR
VAR_IN_OUT
    status : ActivityStatus;
	goToSleep : Process;
	wakeUp : Process;
END_VAR
VAR
    do_request : BOOL := FALSE;
END_VAR

IF status.sleeping THEN
    text := 'Wake up';
    deactivate := wakeUp.statuses.enabledStatus.disabled;
    
    IF do_request THEN
        wakeUp.request();
        do_request := FALSE;
    END_IF

ELSIF status.awake THEN
    text := 'Go to sleep';
    deactivate := goToSleep.statuses.enabledStatus.disabled;
    
    IF do_request THEN
        goToSleep.request();
        do_request := FALSE;
    END_IF
ELSIF status.moving THEN
    text := 'Go to sleep';
    deactivate := TRUE;
    do_request := FALSE;
ELSE
    // we presume the TCS is not initialized yet
    text := 'Wake up';
    deactivate := TRUE;
    do_request := FALSE;
END_IF

END_FUNCTION_BLOCK

// ---- MTCS/Common/Widgets/MeasurementWidget.TcPOU
FUNCTION_BLOCK MeasurementWidget
VAR_INPUT
    value : LREAL;
    actualStatus : STRING;
END_VAR
VAR_IN_OUT
    healthStatus : HealthStatus;
END_VAR
VAR_OUTPUT
    display : STRING;
    _formatString : FB_FormatString;
END_VAR
VAR
    name : STRING;
    actualStatusWidget : StatusWidget;
    format : STRING;
END_VAR

actualStatusWidget(text  := actualStatus,
                   color := HealthToColor(healthStatus));

IF healthStatus.good OR healthStatus.warning THEN
    _formatString(sFormat := format, 
                  arg1    := F_LREAL(value),
                  sOut    => display);
ELSE
    display := '';
END_IF

METHOD FB_init : BOOL
VAR_INPUT
	bInitRetains : BOOL; // if TRUE, the retain variables are initialized (warm start / cold start)
	bInCopyCode : BOOL;  // if TRUE, the instance afterwards gets moved into the copy code (online change)
    n : STRING;
    f : STRING;
END_VAR
name := n;
format := f;
END_METHOD

END_FUNCTION_BLOCK

// ---- MTCS/Common/Widgets/ProcessStepWidget.TcPOU
FUNCTION_BLOCK ProcessStepWidget
VAR_INPUT
    null : BOOL := FALSE;
END_VAR
VAR_IN_OUT
    ref : ProcessStep;
END_VAR
VAR_OUTPUT
	color : StatusColor;
	description : STRING;
	statusText : STRING;
    inivisible : BOOL;
END_VAR
VAR
END_VAR

description := ref.description;
statusText := ref.actualStatus;

IF null THEN
   
    inivisible := TRUE;

ELSIF ref.statuses.enabledStatus.enabled THEN
    
    inivisible := FALSE;
    
    IF ref.isGood() THEN
    
        IF ref.isBusy() THEN
            color.bg := Colors.BLUE;
            color.fg := Colors.WHITE;
        END_IF
        
    ELSIF ref.isWarning() THEN
        
        color.bg := Colors.ORANGE;
        color.bg := Colors.WHITE;
        
    ELSE
        
        color.bg := Colors.RED;
        color.fg := Colors.WHITE;
        
    END_IF

ELSE
    
    inivisible := FALSE;
    
    statusText := '';
    color.bg := Colors.GRAY;
    color.fg := Colors.BLACK;
    
END_IF

END_FUNCTION_BLOCK

// ---- MTCS/Common/Widgets/SimpleRelayWidget.TcPOU
FUNCTION_BLOCK SimpleRelayWidget
VAR_OUTPUT
    text : STRING;
    deactivate : BOOL;
END_VAR
VAR_IN_OUT
    ref : SimpleRelay;
END_VAR
VAR
    do_request : BOOL := FALSE;
END_VAR

IF ref.digitalOutput THEN
    text := 'Disable';
    IF do_request THEN
        ref.setEnabled(enabled := FALSE);
        do_request := FALSE;
	END_IF
ELSE
    text := 'Enable';
    IF do_request THEN
        ref.setEnabled(enabled := TRUE);
        do_request := FALSE;
	END_IF
END_IF
deactivate := ref.processes.setEnabled.statuses.enabledStatus.disabled;

END_FUNCTION_BLOCK

// ---- MTCS/Common/Widgets/SystemButtonWidget.TcPOU
FUNCTION_BLOCK SystemButtonWidget
VAR_INPUT
    color : StatusColor;
END_VAR
VAR_IN_OUT
    activeTab : INT;
END_VAR
VAR_OUTPUT
    name : STRING;
    thisTab : INT;
    activated : BOOL;
    notActivated : BOOL;
    
    isNotGreen : BOOL;
    isNotRed : BOOL;
    isNotBlue : BOOL;
    isNotOrange : BOOL;
    isNotGray : BOOL;
END_VAR
VAR
    do_activate : BOOL;
END_VAR



IF do_activate THEN
    activeTab := thisTab;
    do_activate := FALSE;
END_IF

activated := activeTab = thisTab;
notActivated := NOT activated;

isNotRed    := color.bg <> Colors.RED;
isNotBlue   := color.bg <> Colors.BLUE;
isNotOrange := color.bg <> Colors.ORANGE;
isNotGray   := color.bg <> Colors.GRAY;
isNotGreen  := color.bg <> Colors.GREEN;

METHOD FB_init : BOOL
VAR_INPUT
	bInitRetains : BOOL; // if TRUE, the retain variables are initialized (warm start / cold start)
	bInCopyCode : BOOL;  // if TRUE, the instance afterwards gets moved into the copy code (online change)
    n : STRING;
    tab : INT;
END_VAR
name := n;
thisTab := tab;
END_METHOD

END_FUNCTION_BLOCK

// ---- MTCS/Cover/StateMachines/CoverApertureProcedure.TcPOU
FUNCTION_BLOCK CoverApertureProcedure EXTENDS SM_CoverApertureProcedure
VAR_INPUT
END_VAR
VAR_OUTPUT
END_VAR
VAR
    substate : INT;
    _cause : STRING;
    _ton : TON;
END_VAR

_update();

// run the procedure
CASE state OF
    CoverApertureProcedureStates.IDLE:
        _idle();
    CoverApertureProcedureStates.ABORTED:
        _aborted();
    CoverApertureProcedureStates.PREPARE_PROCESS:
        _prepareProcess();
    CoverApertureProcedureStates.ENABLING_RELAYS:
        _enablingRelays();
    CoverApertureProcedureStates.ENABLING_MOTORS:
        _enablingMotors();
    CoverApertureProcedureStates.OPENING_TOP_PANELS:
        _openingTopPanels();
    CoverApertureProcedureStates.OPENING_BOTH_PANELS:
        _openingBothPanels();
    CoverApertureProcedureStates.ENABLING_MAGNETS:
        _enablingMagnets();
    CoverApertureProcedureStates.DISABLING_MAGNETS:
        _disablingMagnets();
    CoverApertureProcedureStates.CLOSING_BOTTOM_PANELS:
        _closingBottomPanels();
    CoverApertureProcedureStates.CLOSING_BOTH_PANELS:
        _closingBothPanels();
    CoverApertureProcedureStates.DISABLING_MOTORS:
        _disablingMotors();
    CoverApertureProcedureStates.DISABLING_RELAYS:
        _disablingRelays();
    CoverApertureProcedureStates.ABORTING:
        _aborting();
    CoverApertureProcedureStates.RESETTING:
        _resetting();
END_CASE

IF state = CoverApertureProcedureStates.ERROR THEN
    actualStatus := _cause;
ELSE
    actualStatus := _stateToString(state);
END_IF

_update();

METHOD _closingBothPanels
VAR_INPUT
END_VAR
CASE substate OF
    -1:
        // This "special" state will only be active if closing is requested during OPENING_BOTH_PANELS!
        bottom.parts.p1.parts.axis.processes.moveAbsolute.start(
            position    := coverConfig.bottom.p1.closedPosition, 
            maxVelocity := coverConfig.closingVelocity);
        bottom.parts.p2.parts.axis.processes.moveAbsolute.start(
            position    := coverConfig.bottom.p2.closedPosition, 
            maxVelocity := coverConfig.closingVelocity);
        bottom.parts.p3.parts.axis.processes.moveAbsolute.start(
            position    := coverConfig.bottom.p3.closedPosition, 
            maxVelocity := coverConfig.closingVelocity);
        bottom.parts.p4.parts.axis.processes.moveAbsolute.start(
            position    := coverConfig.bottom.p4.closedPosition, 
            maxVelocity := coverConfig.closingVelocity);
        substate := 0;
    0:
        // now also close the top panels
        top.parts.p1.parts.axis.processes.moveAbsolute.start(
            position    := coverConfig.top.p1.closedPosition, 
            maxVelocity := coverConfig.closingVelocity);
        top.parts.p2.parts.axis.processes.moveAbsolute.start(
            position    := coverConfig.top.p2.closedPosition, 
            maxVelocity := coverConfig.closingVelocity);
        top.parts.p3.parts.axis.processes.moveAbsolute.start(
            position    := coverConfig.top.p3.closedPosition, 
            maxVelocity := coverConfig.closingVelocity);
        top.parts.p4.parts.axis.processes.moveAbsolute.start(
            position    := coverConfig.top.p4.closedPosition, 
            maxVelocity := coverConfig.closingVelocity);
        substate := 1;
    1:
        IF top.statuses.healthStatus.bad OR bottom.statuses.healthStatus.bad THEN
            _cause := 'One or more panels in error state!';
            substate := 999; // error!
        ELSIF distance.degrees.value < coverConfig.minDistanceBetweenPanelSets AND NOT bottom.statuses.apertureStatus.closed THEN
            _cause := CONCAT(LREAL_TO_STRING(distance.degrees.value), '° < safety distance!');
            substate := 999; // error!
        ELSIF top.statuses.busyStatus.idle AND bottom.statuses.busyStatus.idle THEN
            IF top.statuses.apertureStatus.closed AND bottom.statuses.apertureStatus.closed THEN
                substate := 1000; // done!
            ELSE
                _cause := 'Panels moved but are not closed!';
                substate := 999; // error!
			END_IF
        END_IF
    999:
        // if there is some error, immediately stop all panels and go to the error state
        top.parts.p1.parts.axis.processes.stop.start();
        top.parts.p2.parts.axis.processes.stop.start();
        top.parts.p3.parts.axis.processes.stop.start();
        top.parts.p4.parts.axis.processes.stop.start();
        bottom.parts.p1.parts.axis.processes.stop.start();
        bottom.parts.p2.parts.axis.processes.stop.start();
        bottom.parts.p3.parts.axis.processes.stop.start();
        bottom.parts.p4.parts.axis.processes.stop.start();
        
        state  := CoverApertureProcedureStates.ERROR;
        substate := 0;
    1000:
        // success, all panels are closed
        substate := 0;
        state    := CoverApertureProcedureStates.DISABLING_MOTORS;
END_CASE
END_METHOD

METHOD _aborted
VAR_INPUT
END_VAR
// not doing anything, just being idle... :-)
;
END_METHOD

METHOD startOpening
VAR_INPUT
END_VAR
IF    state = CoverApertureProcedureStates.IDLE 
   OR state = CoverApertureProcedureStates.ABORTED 
   OR state = CoverApertureProcedureStates.ERROR 
THEN
    state    := CoverApertureProcedureStates.PREPARE_PROCESS;
    substate := 0;
    opening := TRUE;
    closing := FALSE;
ELSIF state = CoverApertureProcedureStates.CLOSING_BOTH_PANELS THEN
    // go to the OPENING_BOTH_PANELS state, but set the substate to the "special" -1 ! 
    substate := -1;
    state := CoverApertureProcedureStates.OPENING_BOTH_PANELS;
    opening := TRUE;
    closing := FALSE;
END_IF

_update();
END_METHOD

METHOD _disablingMotors
VAR_INPUT
END_VAR
CASE substate OF
    0:
        // set the relays of the motors OFF
        top.parts.p1.parts.axis.processes.power.start(enable := FALSE);
        top.parts.p2.parts.axis.processes.power.start(enable := FALSE);
        top.parts.p3.parts.axis.processes.power.start(enable := FALSE);
        top.parts.p4.parts.axis.processes.power.start(enable := FALSE);
        bottom.parts.p1.parts.axis.processes.power.start(enable := FALSE);
        bottom.parts.p2.parts.axis.processes.power.start(enable := FALSE);
        bottom.parts.p3.parts.axis.processes.power.start(enable := FALSE);
        bottom.parts.p4.parts.axis.processes.power.start(enable := FALSE);
        substate := 1;
    1:
        IF      top.parts.p1.parts.axis.processes.power.isIdle()
            AND top.parts.p2.parts.axis.processes.power.isIdle()
            AND top.parts.p3.parts.axis.processes.power.isIdle()
            AND top.parts.p4.parts.axis.processes.power.isIdle()
            AND bottom.parts.p1.parts.axis.processes.power.isIdle()
            AND bottom.parts.p2.parts.axis.processes.power.isIdle()
            AND bottom.parts.p3.parts.axis.processes.power.isIdle()
            AND bottom.parts.p4.parts.axis.processes.power.isIdle()
        THEN
            IF      top.parts.p1.parts.axis.processes.power.isGood()
                AND top.parts.p2.parts.axis.processes.power.isGood()
                AND top.parts.p3.parts.axis.processes.power.isGood()
                AND top.parts.p4.parts.axis.processes.power.isGood()
                AND bottom.parts.p1.parts.axis.processes.power.isGood()
                AND bottom.parts.p2.parts.axis.processes.power.isGood()
                AND bottom.parts.p3.parts.axis.processes.power.isGood()
                AND bottom.parts.p4.parts.axis.processes.power.isGood()
            THEN
                // done!
                state    := CoverApertureProcedureStates.DISABLING_RELAYS;
                substate := 0;
            ELSE
                // error!
                state    := CoverApertureProcedureStates.ERROR;
                substate := 0;
                _cause   := 'Could not disable motors';
            END_IF
		END_IF
END_CASE
END_METHOD

METHOD _prepareProcess
VAR_INPUT
END_VAR
// reset both panelsets
CASE substate OF
    0:
        top.processes.reset.start();
        bottom.processes.reset.start();
        substate := 1;
    1:
        IF top.processes.reset.isIdle() AND bottom.processes.reset.isIdle() THEN
            IF top.processes.reset.isGood() AND bottom.processes.reset.isGood() THEN
                state := CoverApertureProcedureStates.ENABLING_RELAYS;
                substate := 0;
            ELSE
                state    := CoverApertureProcedureStates.ERROR;
                substate := 0;
                _cause   := 'Could not reset panels!';
			END_IF
        END_IF
END_CASE
END_METHOD

METHOD startClosing
VAR_INPUT
END_VAR
IF    state = CoverApertureProcedureStates.IDLE 
   OR state = CoverApertureProcedureStates.ABORTED
   OR state = CoverApertureProcedureStates.ERROR THEN
    state    := CoverApertureProcedureStates.PREPARE_PROCESS;
    substate := 0;
    opening  := FALSE;
    closing  := TRUE;
ELSIF state = CoverApertureProcedureStates.OPENING_BOTH_PANELS THEN
    // go to the CLOSING_BOTH_PANELS state, but set the substate to the "special" -1 ! 
    substate := -1;
    state := CoverApertureProcedureStates.CLOSING_BOTH_PANELS;
    opening  := FALSE;
    closing  := TRUE;
END_IF

_update();
END_METHOD

METHOD _enablingMagnets
VAR_INPUT
END_VAR
CASE substate OF
    0:
        // set the magnets ON
        top.parts.magnetsRelay.processes.setEnabled.start(enabled := TRUE);
        bottom.parts.magnetsRelay.processes.setEnabled.start(enabled := TRUE);
        substate := 1;
    1:
        IF      top.parts.magnetsRelay.processes.setEnabled.isIdle()
            AND bottom.parts.magnetsRelay.processes.setEnabled.isIdle()
        THEN
            IF      top.parts.magnetsRelay.processes.setEnabled.isGood()
                AND bottom.parts.magnetsRelay.processes.setEnabled.isGood()
            THEN
                substate := 2;
            ELSE
                substate := 999; // ERROR!
            END_IF
		END_IF
    2:
        // wait a second or so, to make sure the magnet has done its job of 'locking' the panels.
        // This step may not be strictly needed, but it doesn't hurt to add a small waiting time here...
        _ton(IN := FALSE);
        _ton(IN := TRUE,
             PT := T#3S); 
        substate := 3;
    3:
        _ton(IN := TRUE);
        IF _ton.Q THEN
            substate := 1000; // done!
		END_IF
    999:
        // error!
        state    := CoverApertureProcedureStates.ERROR;
        substate := 0;
        _cause   := 'Could not enable magnets';
    1000:
        // done!
        state    := CoverApertureProcedureStates.DISABLING_MOTORS;
        substate := 0;
END_CASE
END_METHOD

METHOD _disablingRelays
VAR_INPUT
END_VAR
CASE substate OF
    0:
        // set the relays of the motors ON
        top.parts.p1.parts.motorRelay.processes.setEnabled.start(enabled := FALSE);
        top.parts.p2.parts.motorRelay.processes.setEnabled.start(enabled := FALSE);
        top.parts.p3.parts.motorRelay.processes.setEnabled.start(enabled := FALSE);
        top.parts.p4.parts.motorRelay.processes.setEnabled.start(enabled := FALSE);
        bottom.parts.p1.parts.motorRelay.processes.setEnabled.start(enabled := FALSE);
        bottom.parts.p2.parts.motorRelay.processes.setEnabled.start(enabled := FALSE);
        bottom.parts.p3.parts.motorRelay.processes.setEnabled.start(enabled := FALSE);
        bottom.parts.p4.parts.motorRelay.processes.setEnabled.start(enabled := FALSE);
        substate := 1;
    1:
        IF      top.parts.p1.parts.motorRelay.processes.setEnabled.isIdle()
            AND top.parts.p2.parts.motorRelay.processes.setEnabled.isIdle()
            AND top.parts.p3.parts.motorRelay.processes.setEnabled.isIdle()
            AND top.parts.p4.parts.motorRelay.processes.setEnabled.isIdle()
            AND bottom.parts.p1.parts.motorRelay.processes.setEnabled.isIdle()
            AND bottom.parts.p2.parts.motorRelay.processes.setEnabled.isIdle()
            AND bottom.parts.p3.parts.motorRelay.processes.setEnabled.isIdle()
            AND bottom.parts.p4.parts.motorRelay.processes.setEnabled.isIdle()
        THEN
            IF      top.parts.p1.parts.motorRelay.processes.setEnabled.isGood()
                AND top.parts.p2.parts.motorRelay.processes.setEnabled.isGood()
                AND top.parts.p3.parts.motorRelay.processes.setEnabled.isGood()
                AND top.parts.p4.parts.motorRelay.processes.setEnabled.isGood()
                AND bottom.parts.p1.parts.motorRelay.processes.setEnabled.isGood()
                AND bottom.parts.p2.parts.motorRelay.processes.setEnabled.isGood()
                AND bottom.parts.p3.parts.motorRelay.processes.setEnabled.isGood()
                AND bottom.parts.p4.parts.motorRelay.processes.setEnabled.isGood()
            THEN
                substate := 2;
            ELSE
                state    := CoverApertureProcedureStates.ERROR;
                substate := 0;
                _cause   := 'Could not disable relays';
            END_IF
		END_IF
    2:
        // wait a second or so to deal with any transient behaviour
        _ton(IN := FALSE);
        _ton(IN := TRUE,
             PT := T#1S); 
        substate := 3;
    3:
        _ton(IN := TRUE);
        IF _ton.Q THEN
            substate := 4;
		END_IF
    4:
        state    := CoverApertureProcedureStates.IDLE;
        substate := 0;
END_CASE
END_METHOD

METHOD _stateToString : STRING
VAR_INPUT
    x : CoverApertureProcedureStates;
END_VAR
CASE x OF    
    CoverApertureProcedureStates.IDLE:
        _stateToString := 'Idle';
    CoverApertureProcedureStates.ABORTED:
        _stateToString := 'Aborted';
    CoverApertureProcedureStates.PREPARE_PROCESS:
        _stateToString := 'Preparing process';
    CoverApertureProcedureStates.ENABLING_RELAYS:
        _stateToString := 'Enabling relays';
    CoverApertureProcedureStates.ENABLING_MOTORS:
        _stateToString := 'Enabling motors';
    CoverApertureProcedureStates.ENABLING_MAGNETS:
        _stateToString := 'Enabling magnets';
    CoverApertureProcedureStates.DISABLING_RELAYS:
        _stateToString := 'Disabling relays';
    CoverApertureProcedureStates.DISABLING_MOTORS:
        _stateToString := 'Disabling motors';
    CoverApertureProcedureStates.DISABLING_MAGNETS:
        _stateToString := 'Disabling magnets';
    CoverApertureProcedureStates.OPENING_TOP_PANELS:
        _stateToString := 'Opening top panels';
    CoverApertureProcedureStates.OPENING_BOTH_PANELS:
        _stateToString := 'Opening all panels';
    CoverApertureProcedureStates.CLOSING_BOTTOM_PANELS:
        _stateToString := 'Closing bottom panels';
    CoverApertureProcedureStates.CLOSING_BOTH_PANELS:
        _stateToString := 'Closing all panels';
    CoverApertureProcedureStates.ERROR:
        _stateToString := 'Error';
    CoverApertureProcedureStates.RESETTING:
        _stateToString := 'Resetting';
    CoverApertureProcedureStates.ABORTING:
        _stateToString := 'Aborting';
END_CASE
END_METHOD

METHOD _enablingRelays
VAR_INPUT
END_VAR
CASE substate OF
    0:
        // set the relays of the motors ON
        top.parts.p1.parts.motorRelay.processes.setEnabled.start(enabled := TRUE);
        top.parts.p2.parts.motorRelay.processes.setEnabled.start(enabled := TRUE);
        top.parts.p3.parts.motorRelay.processes.setEnabled.start(enabled := TRUE);
        top.parts.p4.parts.motorRelay.processes.setEnabled.start(enabled := TRUE);
        bottom.parts.p1.parts.motorRelay.processes.setEnabled.start(enabled := TRUE);
        bottom.parts.p2.parts.motorRelay.processes.setEnabled.start(enabled := TRUE);
        bottom.parts.p3.parts.motorRelay.processes.setEnabled.start(enabled := TRUE);
        bottom.parts.p4.parts.motorRelay.processes.setEnabled.start(enabled := TRUE);
        substate := 1;
    1:
        IF      top.parts.p1.parts.motorRelay.processes.setEnabled.isIdle()
            AND top.parts.p2.parts.motorRelay.processes.setEnabled.isIdle()
            AND top.parts.p3.parts.motorRelay.processes.setEnabled.isIdle()
            AND top.parts.p4.parts.motorRelay.processes.setEnabled.isIdle()
            AND bottom.parts.p1.parts.motorRelay.processes.setEnabled.isIdle()
            AND bottom.parts.p2.parts.motorRelay.processes.setEnabled.isIdle()
            AND bottom.parts.p3.parts.motorRelay.processes.setEnabled.isIdle()
            AND bottom.parts.p4.parts.motorRelay.processes.setEnabled.isIdle()
        THEN
            IF      top.parts.p1.parts.motorRelay.processes.setEnabled.isGood()
                AND top.parts.p2.parts.motorRelay.processes.setEnabled.isGood()
                AND top.parts.p3.parts.motorRelay.processes.setEnabled.isGood()
                AND top.parts.p4.parts.motorRelay.processes.setEnabled.isGood()
                AND bottom.parts.p1.parts.motorRelay.processes.setEnabled.isGood()
                AND bottom.parts.p2.parts.motorRelay.processes.setEnabled.isGood()
                AND bottom.parts.p3.parts.motorRelay.processes.setEnabled.isGood()
                AND bottom.parts.p4.parts.motorRelay.processes.setEnabled.isGood()
            THEN
                substate := 2;
            ELSE
                state    := CoverApertureProcedureStates.ERROR;
                substate := 0;
                _cause   := 'Could not enable relays';
            END_IF
		END_IF
    2:
        // wait a second or so, to make sure the controllers of the motors are up and running
        _ton(IN := FALSE);
        _ton(IN := TRUE,
             PT := T#1S); 
        substate := 3;
    3:
        _ton(IN := TRUE);
        IF _ton.Q THEN
            substate := 4;
		END_IF
    4:
        state    := CoverApertureProcedureStates.ENABLING_MOTORS;
        substate := 0;
END_CASE
END_METHOD

METHOD _update
VAR_INPUT
END_VAR
SUPER^(top := top, bottom := bottom, coverConfig := coverConfig);

distance(newDegreesValue := ABS(top._maxRelativePosition - bottom._minRelativePosition));
END_METHOD

METHOD _openingBothPanels
VAR_INPUT
END_VAR
CASE substate OF
    -1:
        // This "special" state will only be active if closing is requested during OPENING_BOTH_PANELS!
        top.parts.p1.parts.axis.processes.moveAbsolute.start(
            position    := coverConfig.top.p1.openPosition, 
            maxVelocity := coverConfig.openingVelocity);
        top.parts.p2.parts.axis.processes.moveAbsolute.start(
            position    := coverConfig.top.p2.openPosition, 
            maxVelocity := coverConfig.openingVelocity);
        top.parts.p3.parts.axis.processes.moveAbsolute.start(
            position    := coverConfig.top.p3.openPosition, 
            maxVelocity := coverConfig.openingVelocity);
        top.parts.p4.parts.axis.processes.moveAbsolute.start(
            position    := coverConfig.top.p4.openPosition, 
            maxVelocity := coverConfig.openingVelocity);
        substate := 0;
    0:
        // now also open the bottom panels
        bottom.parts.p1.parts.axis.processes.moveAbsolute.start(
            position    := coverConfig.bottom.p1.openPosition, 
            maxVelocity := coverConfig.openingVelocity);
        bottom.parts.p2.parts.axis.processes.moveAbsolute.start(
            position    := coverConfig.bottom.p2.openPosition, 
            maxVelocity := coverConfig.openingVelocity);
        bottom.parts.p3.parts.axis.processes.moveAbsolute.start(
            position    := coverConfig.bottom.p3.openPosition, 
            maxVelocity := coverConfig.openingVelocity);
        bottom.parts.p4.parts.axis.processes.moveAbsolute.start(
            position    := coverConfig.bottom.p4.openPosition, 
            maxVelocity := coverConfig.openingVelocity);
        substate := 1;
    1:
        IF top.statuses.healthStatus.bad OR bottom.statuses.healthStatus.bad THEN
            _cause := 'One or more panels in error state!';
            substate := 999;
        ELSIF distance.degrees.value < coverConfig.minDistanceBetweenPanelSets AND NOT top.statuses.apertureStatus.open THEN
            _cause := CONCAT(LREAL_TO_STRING(distance.degrees.value), '° < safety distance!');
            substate := 999;
        ELSIF top.statuses.busyStatus.idle AND bottom.statuses.busyStatus.idle THEN
            IF top.statuses.apertureStatus.open AND bottom.statuses.apertureStatus.open THEN
                substate := 1000; // done!
            ELSE
                _cause := 'Panels moved but are not open!';
                substate := 999; // error!
			END_IF
        END_IF
    999:
        // if there is some error, immediately stop all panels and go to the error state
        top.parts.p1.parts.axis.processes.stop.start();
        top.parts.p2.parts.axis.processes.stop.start();
        top.parts.p3.parts.axis.processes.stop.start();
        top.parts.p4.parts.axis.processes.stop.start();
        bottom.parts.p1.parts.axis.processes.stop.start();
        bottom.parts.p2.parts.axis.processes.stop.start();
        bottom.parts.p3.parts.axis.processes.stop.start();
        bottom.parts.p4.parts.axis.processes.stop.start();
        
        state  := CoverApertureProcedureStates.ERROR;
        substate := 0;
    1000:
        // success, all panels are open
        substate := 0;
        state    := CoverApertureProcedureStates.ENABLING_MAGNETS;
END_CASE
END_METHOD

METHOD _aborting
VAR_INPUT
END_VAR
CASE substate OF
    0:  
        // halt all axes
        top.parts.p1.parts.axis.processes.stop.start();
        top.parts.p2.parts.axis.processes.stop.start();
        top.parts.p3.parts.axis.processes.stop.start();
        top.parts.p4.parts.axis.processes.stop.start();
        bottom.parts.p1.parts.axis.processes.stop.start();
        bottom.parts.p2.parts.axis.processes.stop.start();
        bottom.parts.p3.parts.axis.processes.stop.start();
        bottom.parts.p4.parts.axis.processes.stop.start();
        substate := 1;
    1: 
        IF      top.parts.p1.parts.axis.processes.stop.isIdle() 
            AND top.parts.p2.parts.axis.processes.stop.isIdle() 
            AND top.parts.p3.parts.axis.processes.stop.isIdle() 
            AND top.parts.p4.parts.axis.processes.stop.isIdle()
            AND bottom.parts.p2.parts.axis.processes.stop.isIdle() 
            AND bottom.parts.p2.parts.axis.processes.stop.isIdle() 
            AND bottom.parts.p3.parts.axis.processes.stop.isIdle() 
            AND bottom.parts.p4.parts.axis.processes.stop.isIdle() 
        THEN
            // whatever happens, always try to disable the drives
            substate := 2;
        END_IF
    2:
        // disable the drives
        top.parts.p1.parts.axis.processes.power.start(enable := FALSE);
        top.parts.p2.parts.axis.processes.power.start(enable := FALSE);
        top.parts.p3.parts.axis.processes.power.start(enable := FALSE);
        top.parts.p4.parts.axis.processes.power.start(enable := FALSE);
        bottom.parts.p1.parts.axis.processes.power.start(enable := FALSE);
        bottom.parts.p2.parts.axis.processes.power.start(enable := FALSE);
        bottom.parts.p3.parts.axis.processes.power.start(enable := FALSE);
        bottom.parts.p4.parts.axis.processes.power.start(enable := FALSE);
        substate := 3;
    3: 
        IF      top.parts.p1.parts.axis.processes.power.isIdle() 
            AND top.parts.p2.parts.axis.processes.power.isIdle() 
            AND top.parts.p3.parts.axis.processes.power.isIdle() 
            AND top.parts.p4.parts.axis.processes.power.isIdle()
            AND bottom.parts.p2.parts.axis.processes.power.isIdle() 
            AND bottom.parts.p2.parts.axis.processes.power.isIdle() 
            AND bottom.parts.p3.parts.axis.processes.power.isIdle() 
            AND bottom.parts.p4.parts.axis.processes.power.isIdle() 
        THEN
            IF      top.parts.p1.parts.axis.processes.power.isGood() 
                AND top.parts.p2.parts.axis.processes.power.isGood() 
                AND top.parts.p3.parts.axis.processes.power.isGood() 
                AND top.parts.p4.parts.axis.processes.power.isGood()
                AND bottom.parts.p2.parts.axis.processes.power.isGood() 
                AND bottom.parts.p2.parts.axis.processes.power.isGood() 
                AND bottom.parts.p3.parts.axis.processes.power.isGood() 
                AND bottom.parts.p4.parts.axis.processes.power.isGood() 
            THEN
                // Okay, all done!
                state    := CoverApertureProcedureStates.ABORTED;
                substate := 0;
            ELSE
                state    := CoverApertureProcedureStates.ERROR;
                substate := 0;
                _cause   := 'Axes could not be disabled';
            END_IF
        END_IF
            
END_CASE
END_METHOD

METHOD reset
VAR_INPUT
END_VAR
IF state = CoverApertureProcedureStates.ERROR THEN
    // return to the idle state
    state    := CoverApertureProcedureStates.RESETTING;
    substate := 0;
    _cause   := 'RESETTING';
    _update();
END_IF
END_METHOD

METHOD abort
VAR_INPUT
END_VAR
IF statuses.busyStatus.busy THEN
    // go to the aborting state
    state    := CoverApertureProcedureStates.ABORTING;
    substate := 0;
    _cause   := 'ABORTING';
    _update();
END_IF
END_METHOD

METHOD _disablingMagnets
VAR_INPUT
END_VAR
CASE substate OF
    0:
        // set the magnets ON
        top.parts.magnetsRelay.processes.setEnabled.start(enabled := FALSE);
        bottom.parts.magnetsRelay.processes.setEnabled.start(enabled := FALSE);
        substate := 1;
    1:
        IF      top.parts.magnetsRelay.processes.setEnabled.isIdle()
            AND bottom.parts.magnetsRelay.processes.setEnabled.isIdle()
        THEN
            IF      top.parts.magnetsRelay.processes.setEnabled.isGood()
                AND bottom.parts.magnetsRelay.processes.setEnabled.isGood()
            THEN
                substate := 2;
            ELSE
                substate := 999; // ERROR!
                _cause   := 'Could not disable magnets';
            END_IF
		END_IF
    2:
        // wait a few seconds, to make sure the magnet has done its job of 'unlocking' the panels.
        _ton(IN := FALSE);
        _ton(IN := TRUE,
             PT := T#3S); 
        substate := 3;
    3:
        _ton(IN := TRUE);
        IF _ton.Q THEN
            substate := 1000; // done!
		END_IF
    999:
        // error!
        state    := CoverApertureProcedureStates.ERROR;
        substate := 0;
    1000:
        // done!
        state    := CoverApertureProcedureStates.CLOSING_BOTTOM_PANELS;
        substate := 0;
END_CASE
END_METHOD

METHOD _idle
VAR_INPUT
END_VAR
// not doing anything, just being idle... :-)
;
END_METHOD

METHOD _openingTopPanels
VAR_INPUT
END_VAR
CASE substate OF
    0:
        top.parts.p1.parts.axis.processes.moveAbsolute.start(
            position    := coverConfig.top.p1.openPosition, 
            maxVelocity := coverConfig.openingVelocity);
        top.parts.p2.parts.axis.processes.moveAbsolute.start(
            position    := coverConfig.top.p2.openPosition, 
            maxVelocity := coverConfig.openingVelocity);
        top.parts.p3.parts.axis.processes.moveAbsolute.start(
            position    := coverConfig.top.p3.openPosition, 
            maxVelocity := coverConfig.openingVelocity);
        top.parts.p4.parts.axis.processes.moveAbsolute.start(
            position    := coverConfig.top.p4.openPosition, 
            maxVelocity := coverConfig.openingVelocity);
        substate := 1;
    1:
        IF top.statuses.healthStatus.bad THEN
            // if there is some error, immediately stop all panels and go to the error state
            top.parts.p1.parts.axis.processes.stop.start();
            top.parts.p2.parts.axis.processes.stop.start();
            top.parts.p3.parts.axis.processes.stop.start();
            top.parts.p4.parts.axis.processes.stop.start();
            
            state  := CoverApertureProcedureStates.ERROR;
            substate := 0;
            _cause := 'Top panels moving error!';
        ELSE
            IF top.statuses.busyStatus.idle THEN
                // shouldn' t be happening, the top panels should be busy moving!
                top.parts.p1.parts.axis.processes.stop.start();
                top.parts.p2.parts.axis.processes.stop.start();
                top.parts.p3.parts.axis.processes.stop.start();
                top.parts.p4.parts.axis.processes.stop.start();
                state  := CoverApertureProcedureStates.ERROR;
                substate := 0;
                _cause := 'Top panels not busy!';
            ELSE
                IF distance.degrees.value > coverConfig.targetDistanceBetweenPanelSets OR top.statuses.apertureStatus.open THEN
                    // the target distance is reached (or the top panels are fully open), so we can
                    // start opening the bottom panels as well
                    state  := CoverApertureProcedureStates.OPENING_BOTH_PANELS;
                    substate := 0;
                ELSE
                    ; // OK, still moving until the desired distance is reached, nothing to do yet
                END_IF
			END_IF
        END_IF
END_CASE
END_METHOD

METHOD _enablingMotors
VAR_INPUT
END_VAR
CASE substate OF
    0:
        // set the relays of the motors ON
        top.parts.p1.parts.axis.processes.power.start(enable := TRUE);
        top.parts.p2.parts.axis.processes.power.start(enable := TRUE);
        top.parts.p3.parts.axis.processes.power.start(enable := TRUE);
        top.parts.p4.parts.axis.processes.power.start(enable := TRUE);
        bottom.parts.p1.parts.axis.processes.power.start(enable := TRUE);
        bottom.parts.p2.parts.axis.processes.power.start(enable := TRUE);
        bottom.parts.p3.parts.axis.processes.power.start(enable := TRUE);
        bottom.parts.p4.parts.axis.processes.power.start(enable := TRUE);
        substate := 1;
    1:
        IF      top.parts.p1.parts.axis.processes.power.isIdle()
            AND top.parts.p2.parts.axis.processes.power.isIdle()
            AND top.parts.p3.parts.axis.processes.power.isIdle()
            AND top.parts.p4.parts.axis.processes.power.isIdle()
            AND bottom.parts.p1.parts.axis.processes.power.isIdle()
            AND bottom.parts.p2.parts.axis.processes.power.isIdle()
            AND bottom.parts.p3.parts.axis.processes.power.isIdle()
            AND bottom.parts.p4.parts.axis.processes.power.isIdle()
        THEN
            IF      top.parts.p1.parts.axis.processes.power.isGood()
                AND top.parts.p2.parts.axis.processes.power.isGood()
                AND top.parts.p3.parts.axis.processes.power.isGood()
                AND top.parts.p4.parts.axis.processes.power.isGood()
                AND bottom.parts.p1.parts.axis.processes.power.isGood()
                AND bottom.parts.p2.parts.axis.processes.power.isGood()
                AND bottom.parts.p3.parts.axis.processes.power.isGood()
                AND bottom.parts.p4.parts.axis.processes.power.isGood()
            THEN
                IF opening THEN
                    state := CoverApertureProcedureStates.OPENING_TOP_PANELS;
                ELSIF closing THEN
                    state := CoverApertureProcedureStates.DISABLING_MAGNETS;
                ELSE
                    state    := CoverApertureProcedureStates.ERROR;
                    substate := 0;
                    _cause   := 'BUG: not opening or closing';
                END_IF
                substate := 0;
            ELSE
                state    := CoverApertureProcedureStates.ERROR;
                substate := 0;
                _cause   := 'Could not enable motors';
            END_IF
		END_IF
END_CASE
END_METHOD

METHOD _resetting
VAR_INPUT
END_VAR
// reset the axes
CASE substate OF
    0:
        top.parts.p1.parts.axis.processes.reset.start();
        top.parts.p2.parts.axis.processes.reset.start();
        top.parts.p3.parts.axis.processes.reset.start();
        top.parts.p4.parts.axis.processes.reset.start();
        bottom.parts.p1.parts.axis.processes.reset.start();
        bottom.parts.p2.parts.axis.processes.reset.start();
        bottom.parts.p3.parts.axis.processes.reset.start();
        bottom.parts.p4.parts.axis.processes.reset.start();
        substate := 1;
    1:
        IF      top.parts.p1.parts.axis.processes.reset.isIdle() 
            AND top.parts.p2.parts.axis.processes.reset.isIdle() 
            AND top.parts.p3.parts.axis.processes.reset.isIdle() 
            AND top.parts.p4.parts.axis.processes.reset.isIdle() 
            AND bottom.parts.p1.parts.axis.processes.reset.isIdle() 
            AND bottom.parts.p2.parts.axis.processes.reset.isIdle() 
            AND bottom.parts.p3.parts.axis.processes.reset.isIdle() 
            AND bottom.parts.p4.parts.axis.processes.reset.isIdle() 
        THEN
            IF      top.parts.p1.parts.axis.processes.reset.isGood() 
                AND top.parts.p2.parts.axis.processes.reset.isGood() 
                AND top.parts.p3.parts.axis.processes.reset.isGood() 
                AND top.parts.p4.parts.axis.processes.reset.isGood() 
                AND bottom.parts.p1.parts.axis.processes.reset.isGood() 
                AND bottom.parts.p2.parts.axis.processes.reset.isGood() 
                AND bottom.parts.p3.parts.axis.processes.reset.isGood() 
                AND bottom.parts.p4.parts.axis.processes.reset.isGood() 
            THEN
                state    := CoverApertureProcedureStates.IDLE;
                substate := 0;
            ELSE
                state    := CoverApertureProcedureStates.ERROR;
                substate := 0;
                _cause   := 'Could not reset all panels!';
            END_IF
        END_IF
END_CASE
END_METHOD

METHOD _closingBottomPanels
VAR_INPUT
END_VAR
CASE substate OF
    0:
        bottom.parts.p1.parts.axis.processes.moveAbsolute.start(
            position    := coverConfig.bottom.p1.closedPosition, 
            maxVelocity := coverConfig.closingVelocity);
        bottom.parts.p2.parts.axis.processes.moveAbsolute.start(
            position    := coverConfig.bottom.p2.closedPosition, 
            maxVelocity := coverConfig.closingVelocity);
        bottom.parts.p3.parts.axis.processes.moveAbsolute.start(
            position    := coverConfig.bottom.p3.closedPosition, 
            maxVelocity := coverConfig.closingVelocity);
        bottom.parts.p4.parts.axis.processes.moveAbsolute.start(
            position    := coverConfig.bottom.p4.closedPosition, 
            maxVelocity := coverConfig.closingVelocity);
        substate := 1;
    1:
        IF bottom.statuses.healthStatus.bad THEN
            substate := 999; // error!
            _cause := 'Could not close bottom panels!';
        ELSE
            IF bottom.statuses.busyStatus.idle THEN
                // shouldn' t be happening, the top panels should be busy moving!
                substate := 999; // error!
                _cause := 'Bottom panels moving error!';
            ELSE
                IF distance.degrees.value > coverConfig.targetDistanceBetweenPanelSets OR bottom.statuses.apertureStatus.closed THEN
                    // the target distance is reached (or the top panels are fully open), so we can
                    // start opening the bottom panels as well
                    substate := 1000;
                ELSE
                    ; // OK, still moving until the desired distance is reached, nothing to do yet
                END_IF
			END_IF
        END_IF
    999:
        // if there is some error, immediately sbottom all panels and go to the error state
        bottom.parts.p1.parts.axis.processes.stop.start();
        bottom.parts.p2.parts.axis.processes.stop.start();
        bottom.parts.p3.parts.axis.processes.stop.start();
        bottom.parts.p4.parts.axis.processes.stop.start();
        state  := CoverApertureProcedureStates.ERROR;
        substate := 0;
    1000:
        // done!
        state  := CoverApertureProcedureStates.CLOSING_BOTH_PANELS;
        substate := 0;
END_CASE
END_METHOD

END_FUNCTION_BLOCK

// ---- MTCS/Cover/StateMachines/CoverIO.TcPOU
FUNCTION_BLOCK CoverIO EXTENDS SM_CoverIO
VAR_INPUT
END_VAR
VAR_OUTPUT
END_VAR
VAR
    _testVar : INT;
END_VAR

SUPER^();

// do stuff

//SUPER^();

END_FUNCTION_BLOCK

// ---- MTCS/Cover/StateMachines/CoverPanel.TcPOU
FUNCTION_BLOCK CoverPanel EXTENDS SM_CoverPanel
VAR_INPUT
END_VAR
VAR_OUTPUT
END_VAR
VAR
	_relativePosition : LREAL;
END_VAR

SUPER^(
	initializationStatus := initializationStatus, 
	operatingStatus      := operatingStatus, 
	operatorStatus       := operatorStatus, 
	config               := config, 
	coverConfig          := coverConfig);

_relativePosition := parts.axis.actPos.degrees.value - config.closedPosition;

SUPER^(
	initializationStatus := initializationStatus, 
	operatingStatus      := operatingStatus, 
	operatorStatus       := operatorStatus, 
	config               := config, 
	coverConfig          := coverConfig);

END_FUNCTION_BLOCK

// ---- MTCS/Cover/StateMachines/CoverPanelSet.TcPOU
FUNCTION_BLOCK CoverPanelSet EXTENDS SM_CoverPanelSet
VAR_INPUT
END_VAR
VAR_OUTPUT
END_VAR
VAR
	_minRelativePosition : LREAL;	
	_maxRelativePosition : LREAL;	
END_VAR

SUPER^(
	initializationStatus := initializationStatus, 
	operatingStatus      := operatingStatus, 
	operatorStatus       := operatorStatus, 
	config               := config, 
	coverConfig          := coverConfig);

_resetting();


_minRelativePosition := MIN(parts.p1._relativePosition, 
							MIN(parts.p2._relativePosition, 
								MIN(parts.p3._relativePosition, 
									parts.p4._relativePosition)));
_maxRelativePosition := MAX(parts.p1._relativePosition, 
							MAX(parts.p2._relativePosition, 
								MAX(parts.p3._relativePosition, 
									parts.p4._relativePosition)));
									
SUPER^(
	initializationStatus := initializationStatus, 
	operatingStatus      := operatingStatus, 
	operatorStatus       := operatorStatus, 
	config               := config, 
	coverConfig          := coverConfig);

METHOD _resetting
VAR_INPUT
END_VAR
IF processes.reset.statuses.busyStatus.busy THEN
	
	IF processes.reset.statuses.startedStatus.notStarted THEN
		parts.p1.parts.axis.processes.reset.start();
		parts.p2.parts.axis.processes.reset.start();
		parts.p3.parts.axis.processes.reset.start();
		parts.p4.parts.axis.processes.reset.start();
		processes.reset.setStarted();
	END_IF
	
	processes.reset.statuses.healthStatus(
        isGood :=       parts.p1.parts.axis.processes.reset.statuses.healthStatus.good
                    AND parts.p2.parts.axis.processes.reset.statuses.healthStatus.good
                    AND parts.p3.parts.axis.processes.reset.statuses.healthStatus.good
                    AND parts.p4.parts.axis.processes.reset.statuses.healthStatus.good);
	
	processes.reset.statuses.busyStatus(
		isBusy :=       parts.p1.parts.axis.processes.reset.statuses.busyStatus.busy
                    OR  parts.p2.parts.axis.processes.reset.statuses.busyStatus.busy
                    OR  parts.p3.parts.axis.processes.reset.statuses.busyStatus.busy
                    OR  parts.p4.parts.axis.processes.reset.statuses.busyStatus.busy);
ELSE
	processes.reset.setFinished();
END_IF
END_METHOD

END_FUNCTION_BLOCK

// ---- MTCS/Cover/Widgets/CoverIOWidget.TcPOU
FUNCTION_BLOCK CoverIOWidget
VAR_INPUT
END_VAR
VAR_OUTPUT
END_VAR
VAR
	actualStatus : StatusWidget;
	coupler : EtherCatDeviceWidget;
	slot1 : EtherCatDeviceWidget;
	slot2 : EtherCatDeviceWidget;
	slot3 : EtherCatDeviceWidget;
	slot4 : EtherCatDeviceWidget;
	slot5 : EtherCatDeviceWidget;
	slot6 : EtherCatDeviceWidget;
	slot7 : EtherCatDeviceWidget;
	slot8 : EtherCatDeviceWidget;
	slot9 : EtherCatDeviceWidget;
	slot10 : EtherCatDeviceWidget;
	slot11 : EtherCatDeviceWidget;
	slot12 : EtherCatDeviceWidget;
	slot13 : EtherCatDeviceWidget;
END_VAR
VAR_IN_OUT
	io : CoverIO;
END_VAR

actualStatus(text  := io.actualStatus,
             color := HealthToColor(io.statuses.healthStatus));

coupler(device := io.parts.coupler);
slot1(device := io.parts.slot1);
slot2(device := io.parts.slot2);
slot3(device := io.parts.slot3);
slot4(device := io.parts.slot4);
slot5(device := io.parts.slot5);
slot6(device := io.parts.slot6);
slot7(device := io.parts.slot7);
slot8(device := io.parts.slot8);
slot9(device := io.parts.slot9);
slot10(device := io.parts.slot10);
slot11(device := io.parts.slot11);
slot12(device := io.parts.slot12);
slot13(device := io.parts.slot13);

END_FUNCTION_BLOCK

// ---- MTCS/Cover/Widgets/CoverPanelSetWidget.TcPOU
FUNCTION_BLOCK CoverPanelSetWidget
VAR_INPUT
END_VAR
VAR_OUTPUT
    actualStatus : StatusWidget;
END_VAR
VAR_IN_OUT
	panelSet : CoverPanelSet;
	panelSetConfig : CoverPanelSetConfig;
END_VAR
VAR
	p1 : CoverPanelWidget;
	p2 : CoverPanelWidget;
	p3 : CoverPanelWidget;
	p4 : CoverPanelWidget;
    
    magnetsRelay : SimpleRelayWidget;
    
    
    button_p1     : SubSubSystemButtonWidget('Top 1', 0);
    button_p2     : SubSubSystemButtonWidget('Top 2', 1);
    button_p3     : SubSubSystemButtonWidget('Top 3', 2);
    button_p4     : SubSubSystemButtonWidget('Top 4', 3);
    activeTab : INT := 0;
END_VAR

p1(panel := panelSet.parts.p1, panelConfig := panelSetConfig.p1);
p2(panel := panelSet.parts.p2, panelConfig := panelSetConfig.p2);
p3(panel := panelSet.parts.p3, panelConfig := panelSetConfig.p3);
p4(panel := panelSet.parts.p4, panelConfig := panelSetConfig.p4);

magnetsRelay(ref := panelSet.parts.magnetsRelay);

actualStatus(text := panelSet.actualStatus, 
             color := HealthBusyToColor(panelSet.statuses.healthStatus, busyStatus := panelSet.statuses.busyStatus));
             
             
button_p1(color := p1.actualStatus.color, activeTab := activeTab);
button_p2(color := p2.actualStatus.color, activeTab := activeTab);
button_p3(color := p3.actualStatus.color, activeTab := activeTab);
button_p4(color := p4.actualStatus.color, activeTab := activeTab);

END_FUNCTION_BLOCK

// ---- MTCS/Cover/Widgets/CoverPanelWidget.TcPOU
FUNCTION_BLOCK CoverPanelWidget
VAR_INPUT
END_VAR
VAR_OUTPUT
    actualStatus : StatusWidget;
	// percentages
	percentClosed : LREAL;
	percentOpen : LREAL;
	
	drawingRange : LREAL := 251.0; // range of a panel in degrees (according to the drawing)
	drawingAngle : LREAL;
END_VAR
VAR_IN_OUT
	panel : CoverPanel;
	panelConfig : CoverPanelConfig;
END_VAR
VAR
    axis : AngularAxisWidget;
    motorRelay : SimpleRelayWidget;
END_VAR

percentClosed := 100*(panelConfig.openPosition - panel.parts.axis.actPos.degrees.value) 
                 / (panelConfig.openPosition - panelConfig.closedPosition);
percentOpen := 100*(panel.parts.axis.actPos.degrees.value - panelConfig.closedPosition) 
                 / (panelConfig.openPosition - panelConfig.closedPosition);

drawingAngle := - (percentOpen / 100.0 * drawingRange);
			
actualStatus(text := panel.actualStatus, 
             color := HealthBusyToColor(panel.statuses.healthStatus, busyStatus := panel.statuses.busyStatus));

axis(baseRef := panel.parts.axis, ref := panel.parts.axis);

motorRelay(ref := panel.parts.motorRelay);

END_FUNCTION_BLOCK

// ---- MTCS/Cover/Widgets/CoverWidget.TcPOU
FUNCTION_BLOCK CoverWidget
VAR_INPUT
END_VAR
VAR_OUTPUT
	top : CoverPanelSetWidget;
	bottom : CoverPanelSetWidget;
	io : CoverIOWidget;
    configManager : ConfigManagerWidget;
	initializationStatus : InitializationStatusWidget;
	actualStatus : StatusWidget;
	apertureProcedureStatus : StatusWidget;
END_VAR
VAR_IN_OUT
	ref : Cover;
END_VAR
VAR
    activeTab : CoverTabs := CoverTabs.OVERVIEW;
    button_overview   : SubSystemButtonWidget('Overview', CoverTabs.OVERVIEW);
    button_top        : SubSystemButtonWidget('Top'     , CoverTabs.TOP);
    button_bottom     : SubSystemButtonWidget('Bottom'  , CoverTabs.BOTTOM);
    button_io         : SubSystemButtonWidget('I/O'     , CoverTabs.IO);
    button_config     : SubSystemButtonWidget('Config'  , CoverTabs.CONFIG);
    
    button_initialize : InitializeButtonWidget;
    button_operating  : OperatingButtonWidget;
    button_locking    : LockingButtonWidget;
    
    
    activeConfigTab : CoverConfigTabs := CoverConfigTabs.GENERAL;
END_VAR

top(panelSet := ref.parts.top, panelSetConfig := ref.config.top);
bottom(panelSet := ref.parts.bottom, panelSetConfig := ref.config.bottom);
io(io := ref.parts.io);
initializationStatus(status := ref.statuses.initializationStatus);
actualStatus(text  := ref.actualStatus,
             color := SystemToColor(healthStatus := ref.statuses.healthStatus,
                                    busyStatus   := ref.statuses.busyStatus,
                                    initializationStatus := ref.statuses.initializationStatus,
                                    operatingStatus := ref.statuses.operatingStatus));
configManager(mgr := ref.parts.configManager);
apertureProcedureStatus(text := ref.parts.apertureProcedure.actualStatus,
                        color := HealthBusyToColor(healthStatus := ref.parts.apertureProcedure.statuses.healthStatus,
                                                   busyStatus   := ref.parts.apertureProcedure.statuses.busyStatus));

button_overview(    color := actualStatus.color                 , activeTab := activeTab);
button_top(         color := top.actualStatus.color             , activeTab := activeTab);
button_bottom(      color := bottom.actualStatus.color          , activeTab := activeTab);
button_io(          color := io.actualStatus.color              , activeTab := activeTab);
button_config(      color := configManager.actualStatus.color   , activeTab := activeTab);

button_initialize(status := ref.statuses.initializationStatus, process := ref.processes.initialize);
button_operating(status := ref.statuses.operatingStatus, process := ref.processes.changeOperatingState);
button_locking(status := ref.statuses.initializationStatus, lock := ref.processes.lock, unlock := ref.processes.unlock);

END_FUNCTION_BLOCK

// ---- MTCS/Hydraulics/StateMachines/HydraulicsIO.TcPOU
FUNCTION_BLOCK HydraulicsIO EXTENDS SM_HydraulicsIO
VAR_INPUT
END_VAR
VAR_OUTPUT
END_VAR
VAR
END_VAR

SUPER^(safetyIO := safetyIO);

END_FUNCTION_BLOCK

// ---- MTCS/Hydraulics/StateMachines/HydraulicsPumpsGroupIO.TcPOU
FUNCTION_BLOCK HydraulicsPumpsGroupIO EXTENDS SM_HydraulicsPumpsGroupIO
VAR_INPUT
END_VAR
VAR_OUTPUT
END_VAR
VAR
END_VAR

SUPER^();

END_FUNCTION_BLOCK

// ---- MTCS/Hydraulics/StateMachines/HydraulicsSide.TcPOU
FUNCTION_BLOCK HydraulicsSide EXTENDS SM_HydraulicsSide
VAR_INPUT
END_VAR
VAR_OUTPUT
END_VAR
VAR
    isTop : BOOL;
    _resettingDriveState : INT;
    _resettingDriveTon : TON;
END_VAR

_update();

_resettingDrive();
_changingFrequencySetpoint();

// simulation values
IF GLOBAL.config.SIMULATION_ACTIVE THEN
    entranceFilter1OK := TRUE;
    entranceFilter2OK := TRUE;
    entranceFilter3OK := TRUE;
    entranceFilter4OK := TRUE;
END_IF


_update();

METHOD setSide
VAR_INPUT
    top : BOOL;
END_VAR
isTop := top;
END_METHOD

METHOD _resettingDrive
VAR_INPUT
END_VAR
IF processes.resetDrive.isBusy() THEN
    
    // set the signal high for a little while
    CASE _resettingDriveState OF
        0:
            resetDriveSignal := TRUE;
            _resettingDriveTon(IN := FALSE);
            _resettingDriveTon(IN := TRUE,
                               PT := T#500MS); 
            _resettingDriveState := 1;
        1:
            _resettingDriveTon(IN := TRUE);
            IF _resettingDriveTon.Q THEN
                _resettingDriveState := 2;
			END_IF
        2:
            resetDriveSignal := FALSE;
            // wait again a little while
            _resettingDriveTon(IN := FALSE);
            _resettingDriveTon(IN := TRUE,
                               PT := T#500MS); 
            _resettingDriveState := 3;
        3:
            _resettingDriveTon(IN := TRUE);
            IF _resettingDriveTon.Q THEN
                _resettingDriveState := 4;
			END_IF
        4:
            // done!
            processes.resetDrive.setGood();
            processes.resetDrive.setFinished();
            _resettingDriveState := 0;
            
	END_CASE

END_IF
END_METHOD

METHOD _update
VAR_INPUT
END_VAR
// copy some values from the safety
IF isTop THEN
    driveTripOK := safetyHydraulics.topTripOK;
    driveRelease := safetyHydraulics.pumpsRelease;
    driveMinFrequency := safetyHydraulics.pumpsMinFrequency;
ELSE
    driveTripOK := safetyHydraulics.bottomTripOK;
    driveRelease := safetyHydraulics.pumpsRelease;
    driveMinFrequency := safetyHydraulics.pumpsMinFrequency;
END_IF

// update the state machine
SUPER^(
    operatorStatus := operatorStatus, 
    operatingStatus := operatingStatus, 
    safetyHydraulics := safetyHydraulics,
    config := config,
    hydraulicsConfig := hydraulicsConfig);
END_METHOD

METHOD _changingFrequencySetpoint
VAR_INPUT
END_VAR
VAR
    limitedSetpoint : LREAL;
END_VAR
IF processes.changeFrequencySetpoint.isBusy() THEN
    

    // limit the value
    limitedSetpoint := LIMIT(-config.maxFrequency, processes.changeFrequencySetpoint.get.setpoint, config.maxFrequency);
    
    // update the setpoint
    driveSetpoint(newHertzValue := limitedSetpoint);
    
    // update the analog output
    driveSetpointSignal := LREAL_TO_INT(driveSetpoint.hertz.value / 100.0 * (EXPT(2, 15)-1));
    
    // done
    processes.changeFrequencySetpoint.setGood();
    processes.changeFrequencySetpoint.setFinished();
    
END_IF
END_METHOD

END_FUNCTION_BLOCK

// ---- MTCS/Hydraulics/Widgets/HydraulicsSideWidget.TcPOU
FUNCTION_BLOCK HydraulicsSideWidget
VAR_INPUT
    powered : BOOL;
END_VAR
VAR_OUTPUT
	actualStatus : StatusWidget;
	driveStatus : StatusWidget;
	pressureStatus : StatusWidget;
END_VAR
VAR_IN_OUT
    ref : HydraulicsSide;
END_VAR
VAR
    _formatString : FB_FormatString;
    
END_VAR


actualStatus(text  := ref.actualStatus,
             color := HealthBusyToColor(healthStatus := ref.statuses.healthStatus, busyStatus := ref.statuses.busyStatus));
             

// update the driveStatus 
IF NOT powered THEN
   
    driveStatus.color.fg := COLORS.BLACK;
    driveStatus.color.bg := COLORS.GRAY;
    driveStatus.text := 'Powered off';
      
